LIN {X 0,Y 165.63,Z 443.538,A -85,B 0,C 180,E1 -26666.996,E2 -26666.996} C_VEL
LIN {X 0,Y 159.876,Z 456.557,A -85,B 0,C 180,E1 -26668.46,E2 -26668.46} C_VEL
LIN {X 0,Y 153.534,Z 468.796,A -85,B 0,C 180,E1 -26670.356,E2 -26670.356} C_VEL
LIN {X 0,Y 146.219,Z 480.711,A -85,B 0,C 180,E1 -26672.743,E2 -26672.743} C_VEL
LIN {X 0,Y 138.42,Z 491.702,A -85,B 0,C 180,E1 -26675.675,E2 -26675.675} C_VEL
LIN {X 0,Y 131.109,Z 500.936,A -85,B 0,C 180,E1 -26678.992,E2 -26678.992} C_VEL
LIN {X 0,Y 123.678,Z 509.508,A -85,B 0,C 180,E1 -26683.144,E2 -26683.144} C_VEL
LIN {X 0,Y 116.368,Z 517.34,A -85,B 0,C 180,E1 -26688.371,E2 -26688.371} C_VEL
LIN {X 0,Y 109.45,Z 524.137,A -85,B 0,C 180,E1 -26694.699,E2 -26694.699} C_VEL
LIN {X 0,Y 104.079,Z 529.404,A -85,B 0,C 180,E1 -26701.794,E2 -26701.794} C_VEL
LIN {X 0,Y 100.374,Z 533.276,A -85,B 0,C 180,E1 -26709.509,E2 -26709.509} C_VEL
LIN {X 0,Y 98.431,Z 535.839,A -85,B 0,C 180,E1 -26717.633,E2 -26717.633} C_VEL
LIN {X 0,Y 98.114,Z 537.142,A -85,B 0,C 180,E1 -26725.894,E2 -26725.894} C_VEL
LIN {X 0,Y 98.331,Z 537.315,A -85,B 0,C 180,E1 -26730.002,E2 -26730.002} C_VEL
LIN {X 0,Y 98.105,Z 537.113,A -85,B 0,C 180,E1 -26734.272,E2 -26734.272} C_VEL
LIN {X 0,Y 98.447,Z 535.805,A -85,B 0,C 180,E1 -26742.368,E2 -26742.368} C_VEL
LIN {X 0,Y 100.42,Z 533.218,A -85,B 0,C 180,E1 -26750.484,E2 -26750.484} C_VEL
LIN {X 0,Y 100.858,Z 532.685,A -85,B 0,C 180,E1 -26751.673,E2 -26751.673} C_VEL
LIN {X 0,Y 101.579,Z 531.255,A -85,B 0,C 180,E1 -26754.886,E2 -26754.886} C_VEL
LIN {X 0,Y 101.656,Z 528.502,A -85,B 0,C 180,E1 -26760.267,E2 -26760.267} C_VEL
LIN {X 0,Y 102.166,Z 525.971,A -85,B 0,C 180,E1 -26764.5,E2 -26764.5} C_VEL
LIN {X 0,Y 103.612,Z 523.788,A -85,B 0,C 180,E1 -26767.46,E2 -26767.46} C_VEL
LIN {X 0,Y 104.389,Z 523.002,A -85,B 0,C 180,E1 -26768.362,E2 -26768.362} C_VEL
LIN {X 0,Y 112.099,Z 515.87,A -85,B 0,C 180,E1 -26774.856,E2 -26774.856} C_VEL
LIN {X 0,Y 119.581,Z 508.219,A -85,B 0,C 180,E1 -26779.822,E2 -26779.822} C_VEL
LIN {X 0,Y 127.951,Z 498.926,A -85,B 0,C 180,E1 -26784.114,E2 -26784.114} C_VEL
LIN {X 0,Y 135.656,Z 489.398,A -85,B 0,C 180,E1 -26787.339,E2 -26787.339} C_VEL
LIN {X 0,Y 143.86,Z 477.978,A -85,B 0,C 180,E1 -26790.129,E2 -26790.129} C_VEL
LIN {X 0,Y 150.827,Z 466.569,A -85,B 0,C 180,E1 -26792.293,E2 -26792.293} C_VEL
LIN {X 0,Y 157.321,Z 454.193,A -85,B 0,C 180,E1 -26794.033,E2 -26794.033} C_VEL
LIN {X 0,Y 163.247,Z 440.627,A -85,B 0,C 180,E1 -26795.431,E2 -26795.431} C_VEL
LIN {X 0,Y 168.126,Z 426.606,A -85,B 0,C 180,E1 -26796.496,E2 -26796.496} C_VEL
LIN {X 0,Y 171.919,Z 412.179,A -85,B 0,C 180,E1 -26797.272,E2 -26797.272} C_VEL
LIN {X 0,Y 174.531,Z 397.305,A -85,B 0,C 180,E1 -26797.845,E2 -26797.845} C_VEL
LIN {X 0,Y 179.458,Z 349.439,A -85,B 0,C 180,E1 -26799.136,E2 -26799.136} C_VEL
LIN {X 0,Y 179.327,Z 348.411,A -85,B 0,C 180,E1 -26799.347,E2 -26799.347} C_VEL
LIN {X 0,Y 176.957,Z 341.677,A -85,B 0,C 180,E1 -26802.134,E2 -26802.134} C_VEL
LIN {X 0,Y 174.69,Z 335.913,A -85,B 0,C 180,E1 -26805.214,E2 -26805.214} C_VEL
LIN {X 0,Y 173.074,Z 332.046,A -85,B 0,C 180,E1 -26807.84,E2 -26807.84} C_VEL
LIN {X 0,Y 171.759,Z 329.073,A -85,B 0,C 180,E1 -26810.432,E2 -26810.432} C_VEL
LIN {X 0,Y 170.704,Z 326.371,A -85,B 0,C 180,E1 -26813.203,E2 -26813.203} C_VEL
LIN {X 0,Y 169.547,Z 323.722,A -85,B 0,C 180,E1 -26818.219,E2 -26818.219} C_VEL
LIN {X 0,Y 169.402,Z 323.159,A -85,B 0,C 180,E1 -26820,E2 -26820} C_VEL
LIN {X 0,Y 169.554,Z 323.797,A -85,B 0,C 180,E1 -26824.756,E2 -26824.756} C_VEL
LIN {X 0,Y 170.9,Z 326.862,A -85,B 0,C 180,E1 -26830.197,E2 -26830.197} C_VEL
LIN {X 0,Y 172.792,Z 331.172,A -85,B 0,C 180,E1 -26834.386,E2 -26834.386} C_VEL
LIN {X 0,Y 174.529,Z 335.32,A -85,B 0,C 180,E1 -26837.275,E2 -26837.275} C_VEL
LIN {X 0,Y 176.538,Z 340.227,A -85,B 0,C 180,E1 -26840.037,E2 -26840.037} C_VEL
LIN {X 0,Y 179.327,Z 347.998,A -85,B 0,C 180,E1 -26843.329,E2 -26843.329} C_VEL
LIN {X 0,Y 179.502,Z 348.597,A -85,B 0,C 180,E1 -26843.528,E2 -26843.528} C_VEL
LIN {X 0,Y 175.144,Z 392.557,A -85,B 0,C 180,E1 -26844.699,E2 -26844.699} C_VEL
LIN {X 0,Y 172.696,Z 407.451,A -85,B 0,C 180,E1 -26845.285,E2 -26845.285} C_VEL
LIN {X 0,Y 169.623,Z 420.1,A -85,B 0,C 180,E1 -26846.028,E2 -26846.028} C_VEL
LIN {X 0,Y 164.897,Z 434.553,A -85,B 0,C 180,E1 -26847.164,E2 -26847.164} C_VEL
LIN {X 0,Y 159.141,Z 448.284,A -85,B 0,C 180,E1 -26848.631,E2 -26848.631} C_VEL
LIN {X 0,Y 153.259,Z 459.955,A -85,B 0,C 180,E1 -26850.346,E2 -26850.346} C_VEL
LIN {X 0,Y 146.105,Z 471.975,A -85,B 0,C 180,E1 -26852.669,E2 -26852.669} C_VEL
LIN {X 0,Y 138.063,Z 483.246,A -85,B 0,C 180,E1 -26855.465,E2 -26855.465} C_VEL
LIN {X 0,Y 130.537,Z 492.568,A -85,B 0,C 180,E1 -26858.678,E2 -26858.678} C_VEL
LIN {X 0,Y 122.181,Z 501.604,A -85,B 0,C 180,E1 -26862.827,E2 -26862.827} C_VEL
LIN {X 0,Y 114.62,Z 508.971,A -85,B 0,C 180,E1 -26867.586,E2 -26867.586} C_VEL
LIN {X 0,Y 108.945,Z 514.139,A -85,B 0,C 180,E1 -26872.204,E2 -26872.204} C_VEL
LIN {X 0,Y 102.132,Z 519.688,A -85,B 0,C 180,E1 -26878.928,E2 -26878.928} C_VEL
LIN {X 0,Y 98.187,Z 522.898,A -85,B 0,C 180,E1 -26884.565,E2 -26884.565} C_VEL
LIN {X 0,Y 94.287,Z 525.978,A -85,B 0,C 180,E1 -26892.652,E2 -26892.652} C_VEL
LIN {X 0,Y 92.052,Z 527.802,A -85,B 0,C 180,E1 -26901.215,E2 -26901.215} C_VEL
LIN {X 0,Y 91.365,Z 528.414,A -85,B 0,C 180,E1 -26909.998,E2 -26909.998} C_VEL
LIN {X 0,Y 92.006,Z 527.836,A -85,B 0,C 180,E1 -26918.786,E2 -26918.786} C_VEL
LIN {X 0,Y 94.227,Z 526.051,A -85,B 0,C 180,E1 -26927.356,E2 -26927.356} C_VEL
LIN {X 0,Y 98.143,Z 523.004,A -85,B 0,C 180,E1 -26935.444,E2 -26935.444} C_VEL
LIN {X 0,Y 103.601,Z 518.617,A -85,B 0,C 180,E1 -26942.865,E2 -26942.865} C_VEL
LIN {X 0,Y 110.742,Z 512.748,A -85,B 0,C 180,E1 -26949.39,E2 -26949.39} C_VEL
LIN {X 0,Y 117.572,Z 506.34,A -85,B 0,C 180,E1 -26954.495,E2 -26954.495} C_VEL
LIN {X 0,Y 125.598,Z 498.252,A -85,B 0,C 180,E1 -26959.059,E2 -26959.059} C_VEL
LIN {X 0,Y 134.204,Z 488.494,A -85,B 0,C 180,E1 -26962.995,E2 -26962.995} C_VEL
LIN {X 0,Y 141.959,Z 478.341,A -85,B 0,C 180,E1 -26966.019,E2 -26966.019} C_VEL
LIN {X 0,Y 149.557,Z 466.932,A -85,B 0,C 180,E1 -26968.501,E2 -26968.501} C_VEL
LIN {X 0,Y 156.253,Z 454.749,A -85,B 0,C 180,E1 -26970.625,E2 -26970.625} C_VEL
LIN {X 0,Y 161.922,Z 442.664,A -85,B 0,C 180,E1 -26972.168,E2 -26972.168} C_VEL
LIN {X 0,Y 166.986,Z 429.457,A -85,B 0,C 180,E1 -26973.423,E2 -26973.423} C_VEL
LIN {X 0,Y 171.178,Z 415.274,A -85,B 0,C 180,E1 -26974.414,E2 -26974.414} C_VEL
LIN {X 0,Y 174.201,Z 400.761,A -85,B 0,C 180,E1 -26975.152,E2 -26975.152} C_VEL
LIN {X 0,Y 176.229,Z 385.179,A -85,B 0,C 180,E1 -26975.622,E2 -26975.622} C_VEL
LIN {X 0,Y 179.732,Z 348.839,A -85,B 0,C 180,E1 -26976.589,E2 -26976.589} C_VEL
LIN {X 0,Y 177.194,Z 341.617,A -85,B 0,C 180,E1 -26979.561,E2 -26979.561} C_VEL
LIN {X 0,Y 175.174,Z 336.455,A -85,B 0,C 180,E1 -26982.287,E2 -26982.287} C_VEL
LIN {X 0,Y 173.214,Z 331.803,A -85,B 0,C 180,E1 -26985.46,E2 -26985.46} C_VEL
LIN {X 0,Y 172.172,Z 329.574,A -85,B 0,C 180,E1 -26987.488,E2 -26987.488} C_VEL
LIN {X 0,Y 170.897,Z 326.546,A -85,B 0,C 180,E1 -26990.773,E2 -26990.773} C_VEL
LIN {X 0,Y 169.875,Z 324.156,A -85,B 0,C 180,E1 -26995.253,E2 -26995.253} C_VEL
LIN {X 0,Y 169.668,Z 323.599,A -85,B 0,C 180,E1 -26997.626,E2 -26997.626} C_VEL
LIN {X 0,Y 169.698,Z 323.594,A -85,B 0,C 180,E1 -27000.296,E2 -27000.296} C_VEL
LIN {X 0,Y 170.29,Z 325.277,A -85,B 0,C 180,E1 -27004.438,E2 -27004.438} C_VEL
LIN {X 0,Y 171.166,Z 327.18,A -85,B 0,C 180,E1 -27007.372,E2 -27007.372} C_VEL
LIN {X 0,Y 172.943,Z 331.435,A -85,B 0,C 180,E1 -27011.426,E2 -27011.426} C_VEL
LIN {X 0,Y 174.487,Z 335.046,A -85,B 0,C 180,E1 -27014.059,E2 -27014.059} C_VEL
LIN {X 0,Y 176.715,Z 340.576,A -85,B 0,C 180,E1 -27017.205,E2 -27017.205} C_VEL
LIN {X 0,Y 179.259,Z 347.708,A -85,B 0,C 180,E1 -27020.287,E2 -27020.287} C_VEL
LIN {X 0,Y 179.732,Z 349.271,A -85,B 0,C 180,E1 -27020.831,E2 -27020.831} C_VEL
LIN {X 0,Y 174.564,Z 399.199,A -85,B 0,C 180,E1 -27022.187,E2 -27022.187} C_VEL
LIN {X 0,Y 171.726,Z 414.147,A -85,B 0,C 180,E1 -27022.768,E2 -27022.768} C_VEL
LIN {X 0,Y 167.744,Z 428.611,A -85,B 0,C 180,E1 -27023.584,E2 -27023.584} C_VEL
LIN {X 0,Y 162.524,Z 443.079,A -85,B 0,C 180,E1 -27024.76,E2 -27024.76} C_VEL
LIN {X 0,Y 156.61,Z 456.14,A -85,B 0,C 180,E1 -27026.17,E2 -27026.17} C_VEL
LIN {X 0,Y 150.038,Z 468.405,A -85,B 0,C 180,E1 -27027.993,E2 -27027.993} C_VEL
LIN {X 0,Y 142.493,Z 480.341,A -85,B 0,C 180,E1 -27030.333,E2 -27030.333} C_VEL
LIN {X 0,Y 134.362,Z 491.343,A -85,B 0,C 180,E1 -27033.189,E2 -27033.189} C_VEL
LIN {X 0,Y 126.712,Z 500.585,A -85,B 0,C 180,E1 -27036.467,E2 -27036.467} C_VEL
LIN {X 0,Y 118.259,Z 509.78,A -85,B 0,C 180,E1 -27040.975,E2 -27040.975} C_VEL
LIN {X 0,Y 111.092,Z 516.998,A -85,B 0,C 180,E1 -27045.904,E2 -27045.904} C_VEL
LIN {X 0,Y 103.658,Z 523.798,A -85,B 0,C 180,E1 -27052.398,E2 -27052.398} C_VEL
LIN {X 0,Y 97.793,Z 529.066,A -85,B 0,C 180,E1 -27059.8,E2 -27059.8} C_VEL
LIN {X 0,Y 93.682,Z 532.94,A -85,B 0,C 180,E1 -27067.972,E2 -27067.972} C_VEL
LIN {X 0,Y 91.456,Z 535.504,A -85,B 0,C 180,E1 -27076.673,E2 -27076.673} C_VEL
LIN {X 0,Y 91.004,Z 536.808,A -85,B 0,C 180,E1 -27085.573,E2 -27085.573} C_VEL
LIN {X 0,Y 91.223,Z 536.982,A -85,B 0,C 180,E1 -27090.002,E2 -27090.002} C_VEL
LIN {X 0,Y 91.006,Z 536.799,A -85,B 0,C 180,E1 -27094.431,E2 -27094.431} C_VEL
LIN {X 0,Y 91.471,Z 535.469,A -85,B 0,C 180,E1 -27103.328,E2 -27103.328} C_VEL
LIN {X 0,Y 93.942,Z 532.637,A -85,B 0,C 180,E1 -27112.6,E2 -27112.6} C_VEL
LIN {X 0,Y 98.235,Z 528.616,A -85,B 0,C 180,E1 -27120.852,E2 -27120.852} C_VEL
LIN {X 0,Y 104.389,Z 523.002,A -85,B 0,C 180,E1 -27128.362,E2 -27128.362} C_VEL
LIN {X 0,Y 106.483,Z 520.606,A -85,B 0,C 180,E1 -27131.065,E2 -27131.065} C_VEL
LIN {X 0,Y 108.822,Z 516.381,A -85,B 0,C 180,E1 -27135.684,E2 -27135.684} C_VEL
LIN {X 0,Y 111.632,Z 511.724,A -85,B 0,C 180,E1 -27140.005,E2 -27140.005} C_VEL
LIN {X 0,Y 114.344,Z 508.588,A -85,B 0,C 180,E1 -27142.15,E2 -27142.15} C_VEL
LIN {X 0,Y 122.587,Z 500.012,A -85,B 0,C 180,E1 -27146.233,E2 -27146.233} C_VEL
LIN {X 0,Y 130.553,Z 490.711,A -85,B 0,C 180,E1 -27149.466,E2 -27149.466} C_VEL
LIN {X 0,Y 139.016,Z 479.648,A -85,B 0,C 180,E1 -27152.217,E2 -27152.217} C_VEL
LIN {X 0,Y 146.943,Z 467.351,A -85,B 0,C 180,E1 -27154.558,E2 -27154.558} C_VEL
LIN {X 0,Y 153.578,Z 455.24,A -85,B 0,C 180,E1 -27156.24,E2 -27156.24} C_VEL
LIN {X 0,Y 159.655,Z 442.016,A -85,B 0,C 180,E1 -27157.581,E2 -27157.581} C_VEL
LIN {X 0,Y 164.638,Z 428.465,A -85,B 0,C 180,E1 -27158.611,E2 -27158.611} C_VEL
LIN {X 0,Y 168.878,Z 413.351,A -85,B 0,C 180,E1 -27159.419,E2 -27159.419} C_VEL
LIN {X 0,Y 171.751,Z 397.879,A -85,B 0,C 180,E1 -27160.002,E2 -27160.002} C_VEL
LIN {X 0,Y 176.586,Z 352.392,A -85,B 0,C 180,E1 -27161.19,E2 -27161.19} C_VEL
LIN {X 0,Y 174.45,Z 345.846,A -85,B 0,C 180,E1 -27164.071,E2 -27164.071} C_VEL
LIN {X 0,Y 172.065,Z 339.511,A -85,B 0,C 180,E1 -27167.917,E2 -27167.917} C_VEL
LIN {X 0,Y 170.658,Z 336.056,A -85,B 0,C 180,E1 -27170.818,E2 -27170.818} C_VEL
LIN {X 0,Y 169.526,Z 333.041,A -85,B 0,C 180,E1 -27174.051,E2 -27174.051} C_VEL
LIN {X 0,Y 168.609,Z 330.633,A -85,B 0,C 180,E1 -27178.806,E2 -27178.806} C_VEL
LIN {X 0,Y 168.533,Z 330.233,A -85,B 0,C 180,E1 -27180,E2 -27180} C_VEL
LIN {X 0,Y 168.624,Z 330.752,A -85,B 0,C 180,E1 -27184.283,E2 -27184.283} C_VEL
LIN {X 0,Y 169.777,Z 333.605,A -85,B 0,C 180,E1 -27189.531,E2 -27189.531} C_VEL
LIN {X 0,Y 171.5,Z 337.856,A -85,B 0,C 180,E1 -27193.705,E2 -27193.705} C_VEL
LIN {X 0,Y 173.35,Z 342.671,A -85,B 0,C 180,E1 -27196.989,E2 -27196.989} C_VEL
LIN {X 0,Y 175.206,Z 347.777,A -85,B 0,C 180,E1 -27199.681,E2 -27199.681} C_VEL
LIN {X 0,Y 176.615,Z 352.119,A -85,B 0,C 180,E1 -27201.51,E2 -27201.51} C_VEL
LIN {X 0,Y 171.973,Z 396.261,A -85,B 0,C 180,E1 -27202.65,E2 -27202.65} C_VEL
LIN {X 0,Y 169.092,Z 411.279,A -85,B 0,C 180,E1 -27203.27,E2 -27203.27} C_VEL
LIN {X 0,Y 165.171,Z 425.566,A -85,B 0,C 180,E1 -27204.194,E2 -27204.194} C_VEL
LIN {X 0,Y 160.331,Z 438.781,A -85,B 0,C 180,E1 -27205.299,E2 -27205.299} C_VEL
LIN {X 0,Y 154.397,Z 451.68,A -85,B 0,C 180,E1 -27206.707,E2 -27206.707} C_VEL
LIN {X 0,Y 147.791,Z 463.904,A -85,B 0,C 180,E1 -27208.646,E2 -27208.646} C_VEL
LIN {X 0,Y 141.006,Z 474.391,A -85,B 0,C 180,E1 -27210.708,E2 -27210.708} C_VEL
LIN {X 0,Y 132.761,Z 485.257,A -85,B 0,C 180,E1 -27213.512,E2 -27213.512} C_VEL
LIN {X 0,Y 124.974,Z 494.32,A -85,B 0,C 180,E1 -27216.739,E2 -27216.739} C_VEL
LIN {X 0,Y 116.278,Z 503.071,A -85,B 0,C 180,E1 -27220.929,E2 -27220.929} C_VEL
LIN {X 0,Y 109.458,Z 509.315,A -85,B 0,C 180,E1 -27225.066,E2 -27225.066} C_VEL
LIN {X 0,Y 103.435,Z 514.475,A -85,B 0,C 180,E1 -27229.797,E2 -27229.797} C_VEL
LIN {X 0,Y 96.114,Z 520.023,A -85,B 0,C 180,E1 -27236.741,E2 -27236.741} C_VEL
LIN {X 0,Y 91.807,Z 523.233,A -85,B 0,C 180,E1 -27242.656,E2 -27242.656} C_VEL
LIN {X 0,Y 87.54,Z 526.311,A -85,B 0,C 180,E1 -27251.267,E2 -27251.267} C_VEL
LIN {X 0,Y 85.068,Z 528.134,A -85,B 0,C 180,E1 -27260.488,E2 -27260.488} C_VEL
LIN {X 0,Y 84.3,Z 528.746,A -85,B 0,C 180,E1 -27269.998,E2 -27269.998} C_VEL
LIN {X 0,Y 84.994,Z 528.168,A -85,B 0,C 180,E1 -27279.517,E2 -27279.517} C_VEL
LIN {X 0,Y 87.49,Z 526.383,A -85,B 0,C 180,E1 -27288.741,E2 -27288.741} C_VEL
LIN {X 0,Y 91.766,Z 523.338,A -85,B 0,C 180,E1 -27297.354,E2 -27297.354} C_VEL
LIN {X 0,Y 97.719,Z 518.949,A -85,B 0,C 180,E1 -27305.123,E2 -27305.123} C_VEL
LIN {X 0,Y 105.331,Z 513.084,A -85,B 0,C 180,E1 -27311.851,E2 -27311.851} C_VEL
LIN {X 0,Y 112.614,Z 506.677,A -85,B 0,C 180,E1 -27317.029,E2 -27317.029} C_VEL
LIN {X 0,Y 119.808,Z 499.813,A -85,B 0,C 180,E1 -27321.007,E2 -27321.007} C_VEL
LIN {X 0,Y 127.457,Z 491.798,A -85,B 0,C 180,E1 -27324.418,E2 -27324.418} C_VEL
LIN {X 0,Y 135.392,Z 482.257,A -85,B 0,C 180,E1 -27327.51,E2 -27327.51} C_VEL
LIN {X 0,Y 143.696,Z 470.728,A -85,B 0,C 180,E1 -27330.239,E2 -27330.239} C_VEL
LIN {X 0,Y 149.988,Z 460.498,A -85,B 0,C 180,E1 -27332.108,E2 -27332.108} C_VEL
LIN {X 0,Y 156.542,Z 447.881,A -85,B 0,C 180,E1 -27333.88,E2 -27333.88} C_VEL
LIN {X 0,Y 161.735,Z 435.963,A -85,B 0,C 180,E1 -27335.103,E2 -27335.103} C_VEL
LIN {X 0,Y 166.192,Z 423.162,A -85,B 0,C 180,E1 -27336.129,E2 -27336.129} C_VEL
LIN {X 0,Y 169.968,Z 408.622,A -85,B 0,C 180,E1 -27336.989,E2 -27336.989} C_VEL
LIN {X 0,Y 172.529,Z 394.256,A -85,B 0,C 180,E1 -27337.533,E2 -27337.533} C_VEL
LIN {X 0,Y 176.858,Z 352.376,A -85,B 0,C 180,E1 -27338.606,E2 -27338.606} C_VEL
LIN {X 0,Y 174.75,Z 345.892,A -85,B 0,C 180,E1 -27341.448,E2 -27341.448} C_VEL
LIN {X 0,Y 172.472,Z 339.853,A -85,B 0,C 180,E1 -27345.094,E2 -27345.094} C_VEL
LIN {X 0,Y 171.056,Z 336.449,A -85,B 0,C 180,E1 -27347.95,E2 -27347.95} C_VEL
LIN {X 0,Y 169.834,Z 333.379,A -85,B 0,C 180,E1 -27351.346,E2 -27351.346} C_VEL
LIN {X 0,Y 168.939,Z 331.064,A -85,B 0,C 180,E1 -27355.825,E2 -27355.825} C_VEL
LIN {X 0,Y 168.799,Z 330.627,A -85,B 0,C 180,E1 -27357.734,E2 -27357.734} C_VEL
LIN {X 0,Y 168.845,Z 330.755,A -85,B 0,C 180,E1 -27360.596,E2 -27360.596} C_VEL
LIN {X 0,Y 169.404,Z 332.428,A -85,B 0,C 180,E1 -27364.461,E2 -27364.461} C_VEL
LIN {X 0,Y 170.113,Z 334.141,A -85,B 0,C 180,E1 -27366.97,E2 -27366.97} C_VEL
LIN {X 0,Y 171.58,Z 337.97,A -85,B 0,C 180,E1 -27370.62,E2 -27370.62} C_VEL
LIN {X 0,Y 173.094,Z 341.842,A -85,B 0,C 180,E1 -27373.426,E2 -27373.426} C_VEL
LIN {X 0,Y 174.997,Z 346.976,A -85,B 0,C 180,E1 -27376.327,E2 -27376.327} C_VEL
LIN {X 0,Y 176.805,Z 352.535,A -85,B 0,C 180,E1 -27378.75,E2 -27378.75} C_VEL
LIN {X 0,Y 171.814,Z 399.481,A -85,B 0,C 180,E1 -27380.032,E2 -27380.032} C_VEL
LIN {X 0,Y 168.901,Z 414.27,A -85,B 0,C 180,E1 -27380.577,E2 -27380.577} C_VEL
LIN {X 0,Y 164.64,Z 429.218,A -85,B 0,C 180,E1 -27381.396,E2 -27381.396} C_VEL
LIN {X 0,Y 159.681,Z 442.622,A -85,B 0,C 180,E1 -27382.446,E2 -27382.446} C_VEL
LIN {X 0,Y 153.605,Z 455.724,A -85,B 0,C 180,E1 -27383.788,E2 -27383.788} C_VEL
LIN {X 0,Y 146.861,Z 467.937,A -85,B 0,C 180,E1 -27385.511,E2 -27385.511} C_VEL
LIN {X 0,Y 139.023,Z 479.97,A -85,B 0,C 180,E1 -27387.792,E2 -27387.792} C_VEL
LIN {X 0,Y 130.578,Z 490.985,A -85,B 0,C 180,E1 -27390.557,E2 -27390.557} C_VEL
LIN {X 0,Y 122.594,Z 500.236,A -85,B 0,C 180,E1 -27393.776,E2 -27393.776} C_VEL
LIN {X 0,Y 114.196,Z 508.969,A -85,B 0,C 180,E1 -27397.982,E2 -27397.982} C_VEL
LIN {X 0,Y 106.046,Z 516.658,A -85,B 0,C 180,E1 -27403.2,E2 -27403.2} C_VEL
LIN {X 0,Y 98.064,Z 523.459,A -85,B 0,C 180,E1 -27409.837,E2 -27409.837} C_VEL
LIN {X 0,Y 91.665,Z 528.729,A -85,B 0,C 180,E1 -27417.544,E2 -27417.544} C_VEL
LIN {X 0,Y 87.075,Z 532.603,A -85,B 0,C 180,E1 -27426.201,E2 -27426.201} C_VEL
LIN {X 0,Y 84.485,Z 535.168,A -85,B 0,C 180,E1 -27435.551,E2 -27435.551} C_VEL
LIN {X 0,Y 83.899,Z 536.473,A -85,B 0,C 180,E1 -27445.197,E2 -27445.197} C_VEL
LIN {X 0,Y 84.133,Z 536.649,A -85,B 0,C 180,E1 -27450.002,E2 -27450.002} C_VEL
LIN {X 0,Y 83.9,Z 536.464,A -85,B 0,C 180,E1 -27454.807,E2 -27454.807} C_VEL
LIN {X 0,Y 84.501,Z 535.132,A -85,B 0,C 180,E1 -27464.45,E2 -27464.45} C_VEL
LIN {X 0,Y 87.109,Z 532.543,A -85,B 0,C 180,E1 -27473.793,E2 -27473.793} C_VEL
LIN {X 0,Y 91.722,Z 528.594,A -85,B 0,C 180,E1 -27482.559,E2 -27482.559} C_VEL
LIN {X 0,Y 98.26,Z 523.174,A -85,B 0,C 180,E1 -27490.364,E2 -27490.364} C_VEL
LIN {X 0,Y 106.041,Z 516.504,A -85,B 0,C 180,E1 -27496.807,E2 -27496.807} C_VEL
LIN {X 0,Y 114.344,Z 508.588,A -85,B 0,C 180,E1 -27502.15,E2 -27502.15} C_VEL
LIN {X 0,Y 117.141,Z 505.31,A -85,B 0,C 180,E1 -27504.162,E2 -27504.162} C_VEL
LIN {X 0,Y 120.678,Z 499.746,A -85,B 0,C 180,E1 -27507.746,E2 -27507.746} C_VEL
LIN {X 0,Y 124.469,Z 493.764,A -85,B 0,C 180,E1 -27510.974,E2 -27510.974} C_VEL
LIN {X 0,Y 127.526,Z 489.803,A -85,B 0,C 180,E1 -27512.4,E2 -27512.4} C_VEL
LIN {X 0,Y 136.568,Z 478.275,A -85,B 0,C 180,E1 -27515.096,E2 -27515.096} C_VEL
LIN {X 0,Y 144.752,Z 465.749,A -85,B 0,C 180,E1 -27517.293,E2 -27517.293} C_VEL
LIN {X 0,Y 151.616,Z 453.301,A -85,B 0,C 180,E1 -27518.888,E2 -27518.888} C_VEL
LIN {X 0,Y 157.856,Z 439.627,A -85,B 0,C 180,E1 -27520.139,E2 -27520.139} C_VEL
LIN {X 0,Y 162.577,Z 426.731,A -85,B 0,C 180,E1 -27521.02,E2 -27521.02} C_VEL
LIN {X 0,Y 166.588,Z 412.267,A -85,B 0,C 180,E1 -27521.728,E2 -27521.728} C_VEL
LIN {X 0,Y 169.431,Z 396.965,A -85,B 0,C 180,E1 -27522.25,E2 -27522.25} C_VEL
LIN {X 0,Y 173.884,Z 355.821,A -85,B 0,C 180,E1 -27523.313,E2 -27523.313} C_VEL
LIN {X 0,Y 172.125,Z 350.295,A -85,B 0,C 180,E1 -27526.046,E2 -27526.046} C_VEL
LIN {X 0,Y 170.39,Z 345.291,A -85,B 0,C 180,E1 -27529.304,E2 -27529.304} C_VEL
LIN {X 0,Y 169.28,Z 342.309,A -85,B 0,C 180,E1 -27531.946,E2 -27531.946} C_VEL
LIN {X 0,Y 168.467,Z 339.868,A -85,B 0,C 180,E1 -27534.614,E2 -27534.614} C_VEL
LIN {X 0,Y 167.733,Z 337.709,A -85,B 0,C 180,E1 -27538.8,E2 -27538.8} C_VEL
LIN {X 0,Y 167.663,Z 337.292,A -85,B 0,C 180,E1 -27540,E2 -27540} C_VEL
LIN {X 0,Y 167.755,Z 337.788,A -85,B 0,C 180,E1 -27544.194,E2 -27544.194} C_VEL
LIN {X 0,Y 168.713,Z 340.446,A -85,B 0,C 180,E1 -27548.988,E2 -27548.988} C_VEL
LIN {X 0,Y 170.202,Z 344.537,A -85,B 0,C 180,E1 -27552.977,E2 -27552.977} C_VEL
LIN {X 0,Y 172.076,Z 349.751,A -85,B 0,C 180,E1 -27556.537,E2 -27556.537} C_VEL
LIN {X 0,Y 173.931,Z 355.662,A -85,B 0,C 180,E1 -27559.414,E2 -27559.414} C_VEL
LIN {X 0,Y 169.481,Z 396.544,A -85,B 0,C 180,E1 -27560.423,E2 -27560.423} C_VEL
LIN {X 0,Y 166.581,Z 411.332,A -85,B 0,C 180,E1 -27561.006,E2 -27561.006} C_VEL
LIN {X 0,Y 162.78,Z 424.977,A -85,B 0,C 180,E1 -27561.835,E2 -27561.835} C_VEL
LIN {X 0,Y 158.185,Z 437.489,A -85,B 0,C 180,E1 -27562.794,E2 -27562.794} C_VEL
LIN {X 0,Y 152.11,Z 450.684,A -85,B 0,C 180,E1 -27564.144,E2 -27564.144} C_VEL
LIN {X 0,Y 145.867,Z 462.102,A -85,B 0,C 180,E1 -27565.784,E2 -27565.784} C_VEL
LIN {X 0,Y 138.258,Z 473.788,A -85,B 0,C 180,E1 -27567.967,E2 -27567.967} C_VEL
LIN {X 0,Y 130.344,Z 483.981,A -85,B 0,C 180,E1 -27570.378,E2 -27570.378} C_VEL
LIN {X 0,Y 122.165,Z 493.28,A -85,B 0,C 180,E1 -27573.47,E2 -27573.47} C_VEL
LIN {X 0,Y 112.996,Z 502.299,A -85,B 0,C 180,E1 -27577.531,E2 -27577.531} C_VEL
LIN {X 0,Y 104.54,Z 509.658,A -85,B 0,C 180,E1 -27582.31,E2 -27582.31} C_VEL
LIN {X 0,Y 98.128,Z 514.813,A -85,B 0,C 180,E1 -27587.124,E2 -27587.124} C_VEL
LIN {X 0,Y 90.261,Z 520.359,A -85,B 0,C 180,E1 -27594.268,E2 -27594.268} C_VEL
LIN {X 0,Y 85.553,Z 523.567,A -85,B 0,C 180,E1 -27600.468,E2 -27600.468} C_VEL
LIN {X 0,Y 80.862,Z 526.644,A -85,B 0,C 180,E1 -27609.654,E2 -27609.654} C_VEL
LIN {X 0,Y 78.072,Z 528.467,A -85,B 0,C 180,E1 -27619.626,E2 -27619.626} C_VEL
LIN {X 0,Y 77.225,Z 529.078,A -85,B 0,C 180,E1 -27629.998,E2 -27629.998} C_VEL
LIN {X 0,Y 78.014,Z 528.5,A -85,B 0,C 180,E1 -27640.378,E2 -27640.378} C_VEL
LIN {X 0,Y 80.793,Z 526.716,A -85,B 0,C 180,E1 -27650.36,E2 -27650.36} C_VEL
LIN {X 0,Y 85.515,Z 523.67,A -85,B 0,C 180,E1 -27659.543,E2 -27659.543} C_VEL
LIN {X 0,Y 92.011,Z 519.282,A -85,B 0,C 180,E1 -27667.663,E2 -27667.663} C_VEL
LIN {X 0,Y 100.136,Z 513.42,A -85,B 0,C 180,E1 -27674.572,E2 -27674.572} C_VEL
LIN {X 0,Y 108.02,Z 506.916,A -85,B 0,C 180,E1 -27679.857,E2 -27679.857} C_VEL
LIN {X 0,Y 116.797,Z 498.936,A -85,B 0,C 180,E1 -27684.321,E2 -27684.321} C_VEL
LIN {X 0,Y 126.185,Z 489.2,A -85,B 0,C 180,E1 -27688.139,E2 -27688.139} C_VEL
LIN {X 0,Y 134.554,Z 479.072,A -85,B 0,C 180,E1 -27691.027,E2 -27691.027} C_VEL
LIN {X 0,Y 142.496,Z 467.975,A -85,B 0,C 180,E1 -27693.31,E2 -27693.31} C_VEL
LIN {X 0,Y 149.814,Z 455.577,A -85,B 0,C 180,E1 -27695.351,E2 -27695.351} C_VEL
LIN {X 0,Y 155.822,Z 443.569,A -85,B 0,C 180,E1 -27696.772,E2 -27696.772} C_VEL
LIN {X 0,Y 161.543,Z 429.372,A -85,B 0,C 180,E1 -27697.999,E2 -27697.999} C_VEL
LIN {X 0,Y 165.974,Z 414.934,A -85,B 0,C 180,E1 -27698.909,E2 -27698.909} C_VEL
LIN {X 0,Y 169.028,Z 400.886,A -85,B 0,C 180,E1 -27699.558,E2 -27699.558} C_VEL
LIN {X 0,Y 171.273,Z 384.215,A -85,B 0,C 180,E1 -27700.006,E2 -27700.006} C_VEL
LIN {X 0,Y 174.184,Z 355.781,A -85,B 0,C 180,E1 -27700.729,E2 -27700.729} C_VEL
LIN {X 0,Y 172.281,Z 349.813,A -85,B 0,C 180,E1 -27703.712,E2 -27703.712} C_VEL
LIN {X 0,Y 170.483,Z 344.736,A -85,B 0,C 180,E1 -27707.176,E2 -27707.176} C_VEL
LIN {X 0,Y 168.886,Z 340.389,A -85,B 0,C 180,E1 -27711.59,E2 -27711.59} C_VEL
LIN {X 0,Y 168.071,Z 338.153,A -85,B 0,C 180,E1 -27715.803,E2 -27715.803} C_VEL
LIN {X 0,Y 167.935,Z 337.725,A -85,B 0,C 180,E1 -27717.601,E2 -27717.601} C_VEL
LIN {X 0,Y 167.976,Z 337.835,A -85,B 0,C 180,E1 -27720.599,E2 -27720.599} C_VEL
LIN {X 0,Y 168.587,Z 339.766,A -85,B 0,C 180,E1 -27724.782,E2 -27724.782} C_VEL
LIN {X 0,Y 169.101,Z 341.329,A -85,B 0,C 180,E1 -27726.712,E2 -27726.712} C_VEL
LIN {X 0,Y 170.252,Z 344.508,A -85,B 0,C 180,E1 -27729.804,E2 -27729.804} C_VEL
LIN {X 0,Y 171.566,Z 348.184,A -85,B 0,C 180,E1 -27732.494,E2 -27732.494} C_VEL
LIN {X 0,Y 173.345,Z 353.543,A -85,B 0,C 180,E1 -27735.482,E2 -27735.482} C_VEL
LIN {X 0,Y 174.133,Z 356.068,A -85,B 0,C 180,E1 -27736.655,E2 -27736.655} C_VEL
LIN {X 0,Y 169.349,Z 399.51,A -85,B 0,C 180,E1 -27737.795,E2 -27737.795} C_VEL
LIN {X 0,Y 166.34,Z 414.353,A -85,B 0,C 180,E1 -27738.312,E2 -27738.312} C_VEL
LIN {X 0,Y 162.182,Z 428.694,A -85,B 0,C 180,E1 -27739.057,E2 -27739.057} C_VEL
LIN {X 0,Y 157.105,Z 442.164,A -85,B 0,C 180,E1 -27740.05,E2 -27740.05} C_VEL
LIN {X 0,Y 150.863,Z 455.306,A -85,B 0,C 180,E1 -27741.302,E2 -27741.302} C_VEL
LIN {X 0,Y 144.057,Z 467.329,A -85,B 0,C 180,E1 -27742.9,E2 -27742.9} C_VEL
LIN {X 0,Y 135.836,Z 479.599,A -85,B 0,C 180,E1 -27745.123,E2 -27745.123} C_VEL
LIN {X 0,Y 127.087,Z 490.627,A -85,B 0,C 180,E1 -27747.776,E2 -27747.776} C_VEL
LIN {X 0,Y 118.755,Z 499.887,A -85,B 0,C 180,E1 -27750.898,E2 -27750.898} C_VEL
LIN {X 0,Y 110.875,Z 507.726,A -85,B 0,C 180,E1 -27754.514,E2 -27754.514} C_VEL
LIN {X 0,Y 103.539,Z 514.322,A -85,B 0,C 180,E1 -27758.688,E2 -27758.688} C_VEL
LIN {X 0,Y 94.695,Z 521.569,A -85,B 0,C 180,E1 -27765.168,E2 -27765.168} C_VEL
LIN {X 0,Y 87.282,Z 527.215,A -85,B 0,C 180,E1 -27772.853,E2 -27772.853} C_VEL
LIN {X 0,Y 82.898,Z 530.499,A -85,B 0,C 180,E1 -27779.427,E2 -27779.427} C_VEL
LIN {X 0,Y 78.742,Z 533.707,A -85,B 0,C 180,E1 -27789.085,E2 -27789.085} C_VEL
LIN {X 0,Y 76.928,Z 535.642,A -85,B 0,C 180,E1 -27799.474,E2 -27799.474} C_VEL
LIN {X 0,Y 76.79,Z 536.139,A -85,B 0,C 180,E1 -27804.751,E2 -27804.751} C_VEL
LIN {X 0,Y 77.047,Z 536.316,A -85,B 0,C 180,E1 -27810.002,E2 -27810.002} C_VEL
LIN {X 0,Y 76.793,Z 536.13,A -85,B 0,C 180,E1 -27815.253,E2 -27815.253} C_VEL
LIN {X 0,Y 77.573,Z 534.795,A -85,B 0,C 180,E1 -27825.773,E2 -27825.773} C_VEL
LIN {X 0,Y 80.599,Z 532.206,A -85,B 0,C 180,E1 -27835.85,E2 -27835.85} C_VEL
LIN {X 0,Y 85.67,Z 528.305,A -85,B 0,C 180,E1 -27845.049,E2 -27845.049} C_VEL
LIN {X 0,Y 92.675,Z 523.003,A -85,B 0,C 180,E1 -27853.042,E2 -27853.042} C_VEL
LIN {X 0,Y 101.264,Z 516.161,A -85,B 0,C 180,E1 -27859.769,E2 -27859.769} C_VEL
LIN {X 0,Y 109.317,Z 508.933,A -85,B 0,C 180,E1 -27864.706,E2 -27864.706} C_VEL
LIN {X 0,Y 117.395,Z 501.029,A -85,B 0,C 180,E1 -27868.551,E2 -27868.551} C_VEL
LIN {X 0,Y 125.662,Z 491.994,A -85,B 0,C 180,E1 -27871.748,E2 -27871.748} C_VEL
LIN {X 0,Y 127.526,Z 489.803,A -85,B 0,C 180,E1 -27872.4,E2 -27872.4} C_VEL
LIN {X 0,Y 130.56,Z 485.712,A -85,B 0,C 180,E1 -27873.738,E2 -27873.738} C_VEL
LIN {X 0,Y 134.41,Z 478.89,A -85,B 0,C 180,E1 -27876.383,E2 -27876.383} C_VEL
LIN {X 0,Y 138.22,Z 471.768,A -85,B 0,C 180,E1 -27878.777,E2 -27878.777} C_VEL
LIN {X 0,Y 141.066,Z 467.061,A -85,B 0,C 180,E1 -27879.715,E2 -27879.715} C_VEL
LIN {X 0,Y 148.409,Z 454.388,A -85,B 0,C 180,E1 -27881.283,E2 -27881.283} C_VEL
LIN {X 0,Y 154.783,Z 441.075,A -85,B 0,C 180,E1 -27882.462,E2 -27882.462} C_VEL
LIN {X 0,Y 159.998,Z 427.387,A -85,B 0,C 180,E1 -27883.361,E2 -27883.361} C_VEL
LIN {X 0,Y 164.173,Z 412.97,A -85,B 0,C 180,E1 -27884.022,E2 -27884.022} C_VEL
LIN {X 0,Y 166.985,Z 398.735,A -85,B 0,C 180,E1 -27884.516,E2 -27884.516} C_VEL
LIN {X 0,Y 171.416,Z 359.622,A -85,B 0,C 180,E1 -27885.457,E2 -27885.457} C_VEL
LIN {X 0,Y 169.854,Z 354.388,A -85,B 0,C 180,E1 -27888.363,E2 -27888.363} C_VEL
LIN {X 0,Y 168.539,Z 350.141,A -85,B 0,C 180,E1 -27891.457,E2 -27891.457} C_VEL
LIN {X 0,Y 167.421,Z 346.721,A -85,B 0,C 180,E1 -27895.184,E2 -27895.184} C_VEL
LIN {X 0,Y 166.806,Z 344.612,A -85,B 0,C 180,E1 -27899.397,E2 -27899.397} C_VEL
LIN {X 0,Y 166.785,Z 344.594,A -85,B 0,C 180,E1 -27903.009,E2 -27903.009} C_VEL
LIN {X 0,Y 167.029,Z 345.564,A -85,B 0,C 180,E1 -27905.493,E2 -27905.493} C_VEL
LIN {X 0,Y 167.689,Z 347.484,A -85,B 0,C 180,E1 -27908.587,E2 -27908.587} C_VEL
LIN {X 0,Y 168.905,Z 351.087,A -85,B 0,C 180,E1 -27912.163,E2 -27912.163} C_VEL
LIN {X 0,Y 170.554,Z 356.156,A -85,B 0,C 180,E1 -27915.626,E2 -27915.626} C_VEL
LIN {X 0,Y 171.456,Z 359.288,A -85,B 0,C 180,E1 -27917.231,E2 -27917.231} C_VEL
LIN {X 0,Y 167.233,Z 396.94,A -85,B 0,C 180,E1 -27918.138,E2 -27918.138} C_VEL
LIN {X 0,Y 164.293,Z 411.533,A -85,B 0,C 180,E1 -27918.677,E2 -27918.677} C_VEL
LIN {X 0,Y 160.289,Z 425.511,A -85,B 0,C 180,E1 -27919.492,E2 -27919.492} C_VEL
LIN {X 0,Y 155.584,Z 437.959,A -85,B 0,C 180,E1 -27920.394,E2 -27920.394} C_VEL
LIN {X 0,Y 149.351,Z 451.107,A -85,B 0,C 180,E1 -27921.662,E2 -27921.662} C_VEL
LIN {X 0,Y 142.685,Z 462.9,A -85,B 0,C 180,E1 -27923.293,E2 -27923.293} C_VEL
LIN {X 0,Y 134.332,Z 475.137,A -85,B 0,C 180,E1 -27925.512,E2 -27925.512} C_VEL
LIN {X 0,Y 126.904,Z 484.346,A -85,B 0,C 180,E1 -27927.614,E2 -27927.614} C_VEL
LIN {X 0,Y 118.405,Z 493.635,A -85,B 0,C 180,E1 -27930.609,E2 -27930.609} C_VEL
LIN {X 0,Y 108.813,Z 502.646,A -85,B 0,C 180,E1 -27934.562,E2 -27934.562} C_VEL
LIN {X 0,Y 99.889,Z 510.001,A -85,B 0,C 180,E1 -27939.289,E2 -27939.289} C_VEL
LIN {X 0,Y 93.057,Z 515.151,A -85,B 0,C 180,E1 -27944.152,E2 -27944.152} C_VEL
LIN {X 0,Y 84.604,Z 520.695,A -85,B 0,C 180,E1 -27951.462,E2 -27951.462} C_VEL
LIN {X 0,Y 79.449,Z 523.901,A -85,B 0,C 180,E1 -27957.942,E2 -27957.942} C_VEL
LIN {X 0,Y 74.24,Z 526.977,A -85,B 0,C 180,E1 -27967.747,E2 -27967.747} C_VEL
LIN {X 0,Y 71.114,Z 528.8,A -85,B 0,C 180,E1 -27978.598,E2 -27978.598} C_VEL
LIN {X 0,Y 70.138,Z 529.41,A -85,B 0,C 180,E1 -27989.998,E2 -27989.998} C_VEL
LIN {X 0,Y 71.048,Z 528.833,A -85,B 0,C 180,E1 -28001.408,E2 -28001.408} C_VEL
LIN {X 0,Y 74.183,Z 527.048,A -85,B 0,C 180,E1 -28012.267,E2 -28012.267} C_VEL
LIN {X 0,Y 79.413,Z 524.003,A -85,B 0,C 180,E1 -28022.07,E2 -28022.07} C_VEL
LIN {X 0,Y 86.511,Z 519.614,A -85,B 0,C 180,E1 -28030.532,E2 -28030.532} C_VEL
LIN {X 0,Y 95.177,Z 513.757,A -85,B 0,C 180,E1 -28037.593,E2 -28037.593} C_VEL
LIN {X 0,Y 103.579,Z 507.254,A -85,B 0,C 180,E1 -28042.866,E2 -28042.866} C_VEL
LIN {X 0,Y 112.812,Z 499.277,A -85,B 0,C 180,E1 -28047.245,E2 -28047.245} C_VEL
LIN {X 0,Y 122.594,Z 489.551,A -85,B 0,C 180,E1 -28050.952,E2 -28050.952} C_VEL
LIN {X 0,Y 131.272,Z 479.436,A -85,B 0,C 180,E1 -28053.731,E2 -28053.731} C_VEL
LIN {X 0,Y 138.759,Z 469.352,A -85,B 0,C 180,E1 -28055.735,E2 -28055.735} C_VEL
LIN {X 0,Y 146.244,Z 457.327,A -85,B 0,C 180,E1 -28057.677,E2 -28057.677} C_VEL
LIN {X 0,Y 153.173,Z 444.014,A -85,B 0,C 180,E1 -28059.2,E2 -28059.2} C_VEL
LIN {X 0,Y 159.034,Z 429.893,A -85,B 0,C 180,E1 -28060.357,E2 -28060.357} C_VEL
LIN {X 0,Y 163.55,Z 415.632,A -85,B 0,C 180,E1 -28061.214,E2 -28061.214} C_VEL
LIN {X 0,Y 166.714,Z 401.588,A -85,B 0,C 180,E1 -28061.845,E2 -28061.845} C_VEL
LIN {X 0,Y 168.985,Z 385.496,A -85,B 0,C 180,E1 -28062.259,E2 -28062.259} C_VEL
LIN {X 0,Y 171.723,Z 359.479,A -85,B 0,C 180,E1 -28062.912,E2 -28062.912} C_VEL
LIN {X 0,Y 170.335,Z 354.879,A -85,B 0,C 180,E1 -28065.466,E2 -28065.466} C_VEL
LIN {X 0,Y 168.966,Z 350.519,A -85,B 0,C 180,E1 -28068.605,E2 -28068.605} C_VEL
LIN {X 0,Y 167.76,Z 347.051,A -85,B 0,C 180,E1 -28072.477,E2 -28072.477} C_VEL
LIN {X 0,Y 167.141,Z 345.077,A -85,B 0,C 180,E1 -28076.383,E2 -28076.383} C_VEL
LIN {X 0,Y 167.08,Z 344.741,A -85,B 0,C 180,E1 -28080,E2 -28080} C_VEL
LIN {X 0,Y 167.573,Z 346.601,A -85,B 0,C 180,E1 -28084.209,E2 -28084.209} C_VEL
LIN {X 0,Y 168.024,Z 348.145,A -85,B 0,C 180,E1 -28086.153,E2 -28086.153} C_VEL
LIN {X 0,Y 169.023,Z 351.243,A -85,B 0,C 180,E1 -28089.136,E2 -28089.136} C_VEL
LIN {X 0,Y 170.12,Z 354.632,A -85,B 0,C 180,E1 -28091.618,E2 -28091.618} C_VEL
LIN {X 0,Y 171.677,Z 359.862,A -85,B 0,C 180,E1 -28094.521,E2 -28094.521} C_VEL
LIN {X 0,Y 167.199,Z 399.273,A -85,B 0,C 180,E1 -28095.49,E2 -28095.49} C_VEL
LIN {X 0,Y 164.127,Z 414.148,A -85,B 0,C 180,E1 -28095.97,E2 -28095.97} C_VEL
LIN {X 0,Y 160.004,Z 428.172,A -85,B 0,C 180,E1 -28096.653,E2 -28096.653} C_VEL
LIN {X 0,Y 154.81,Z 441.706,A -85,B 0,C 180,E1 -28097.576,E2 -28097.576} C_VEL
LIN {X 0,Y 148.424,Z 454.89,A -85,B 0,C 180,E1 -28098.74,E2 -28098.74} C_VEL
LIN {X 0,Y 141.112,Z 467.43,A -85,B 0,C 180,E1 -28100.31,E2 -28100.31} C_VEL
LIN {X 0,Y 132.951,Z 479.227,A -85,B 0,C 180,E1 -28102.325,E2 -28102.325} C_VEL
LIN {X 0,Y 123.911,Z 490.267,A -85,B 0,C 180,E1 -28104.844,E2 -28104.844} C_VEL
LIN {X 0,Y 115.23,Z 499.536,A -85,B 0,C 180,E1 -28107.83,E2 -28107.83} C_VEL
LIN {X 0,Y 105.754,Z 508.444,A -85,B 0,C 180,E1 -28111.928,E2 -28111.928} C_VEL
LIN {X 0,Y 96.766,Z 515.976,A -85,B 0,C 180,E1 -28116.977,E2 -28116.977} C_VEL
LIN {X 0,Y 87.56,Z 522.782,A -85,B 0,C 180,E1 -28123.752,E2 -28123.752} C_VEL
LIN {X 0,Y 79.932,Z 528.056,A -85,B 0,C 180,E1 -28132.017,E2 -28132.017} C_VEL
LIN {X 0,Y 74.176,Z 531.932,A -85,B 0,C 180,E1 -28141.726,E2 -28141.726} C_VEL
LIN {X 0,Y 70.69,Z 534.496,A -85,B 0,C 180,E1 -28152.649,E2 -28152.649} C_VEL
LIN {X 0,Y 69.691,Z 535.804,A -85,B 0,C 180,E1 -28164.214,E2 -28164.214} C_VEL
LIN {X 0,Y 69.948,Z 535.983,A -85,B 0,C 180,E1 -28170.002,E2 -28170.002} C_VEL
LIN {X 0,Y 69.925,Z 535.285,A -85,B 0,C 180,E1 -28181.598,E2 -28181.598} C_VEL
LIN {X 0,Y 72.111,Z 533.321,A -85,B 0,C 180,E1 -28192.947,E2 -28192.947} C_VEL
LIN {X 0,Y 76.815,Z 530.088,A -85,B 0,C 180,E1 -28203.297,E2 -28203.297} C_VEL
LIN {X 0,Y 83.529,Z 525.5,A -85,B 0,C 180,E1 -28212.309,E2 -28212.309} C_VEL
LIN {X 0,Y 91.987,Z 519.443,A -85,B 0,C 180,E1 -28219.821,E2 -28219.821} C_VEL
LIN {X 0,Y 100.488,Z 512.777,A -85,B 0,C 180,E1 -28225.265,E2 -28225.265} C_VEL
LIN {X 0,Y 109.652,Z 504.664,A -85,B 0,C 180,E1 -28229.915,E2 -28229.915} C_VEL
LIN {X 0,Y 118.101,Z 496.346,A -85,B 0,C 180,E1 -28233.206,E2 -28233.206} C_VEL
LIN {X 0,Y 126.894,Z 486.49,A -85,B 0,C 180,E1 -28236.044,E2 -28236.044} C_VEL
LIN {X 0,Y 135.983,Z 474.66,A -85,B 0,C 180,E1 -28238.481,E2 -28238.481} C_VEL
LIN {X 0,Y 141.066,Z 467.061,A -85,B 0,C 180,E1 -28239.715,E2 -28239.715} C_VEL
LIN {X 0,Y 143.816,Z 462.306,A -85,B 0,C 180,E1 -28240.586,E2 -28240.586} C_VEL
LIN {X 0,Y 147.22,Z 454.421,A -85,B 0,C 180,E1 -28242.541,E2 -28242.541} C_VEL
LIN {X 0,Y 150.371,Z 446.305,A -85,B 0,C 180,E1 -28244.338,E2 -28244.338} C_VEL
LIN {X 0,Y 152.578,Z 441.046,A -85,B 0,C 180,E1 -28244.983,E2 -28244.983} C_VEL
LIN {X 0,Y 157.695,Z 427.981,A -85,B 0,C 180,E1 -28245.774,E2 -28245.774} C_VEL
LIN {X 0,Y 162.159,Z 413.052,A -85,B 0,C 180,E1 -28246.414,E2 -28246.414} C_VEL
LIN {X 0,Y 165.256,Z 397.561,A -85,B 0,C 180,E1 -28246.892,E2 -28246.892} C_VEL
LIN {X 0,Y 169.16,Z 363.43,A -85,B 0,C 180,E1 -28247.707,E2 -28247.707} C_VEL
LIN {X 0,Y 167.761,Z 358.372,A -85,B 0,C 180,E1 -28250.962,E2 -28250.962} C_VEL
LIN {X 0,Y 166.88,Z 355.401,A -85,B 0,C 180,E1 -28253.653,E2 -28253.653} C_VEL
LIN {X 0,Y 166.393,Z 353.563,A -85,B 0,C 180,E1 -28255.762,E2 -28255.762} C_VEL
LIN {X 0,Y 165.938,Z 351.683,A -85,B 0,C 180,E1 -28259.394,E2 -28259.394} C_VEL
LIN {X 0,Y 165.918,Z 351.663,A -85,B 0,C 180,E1 -28263.024,E2 -28263.024} C_VEL
LIN {X 0,Y 166.239,Z 353.024,A -85,B 0,C 180,E1 -28266.067,E2 -28266.067} C_VEL
LIN {X 0,Y 166.678,Z 354.482,A -85,B 0,C 180,E1 -28268.182,E2 -28268.182} C_VEL
LIN {X 0,Y 167.694,Z 357.799,A -85,B 0,C 180,E1 -28271.473,E2 -28271.473} C_VEL
LIN {X 0,Y 169.233,Z 363.146,A -85,B 0,C 180,E1 -28275.023,E2 -28275.023} C_VEL
LIN {X 0,Y 165.373,Z 396.671,A -85,B 0,C 180,E1 -28275.771,E2 -28275.771} C_VEL
LIN {X 0,Y 162.419,Z 411.246,A -85,B 0,C 180,E1 -28276.272,E2 -28276.272} C_VEL
LIN {X 0,Y 158.47,Z 424.924,A -85,B 0,C 180,E1 -28277.004,E2 -28277.004} C_VEL
LIN {X 0,Y 153.264,Z 438.425,A -85,B 0,C 180,E1 -28277.916,E2 -28277.916} C_VEL
LIN {X 0,Y 146.888,Z 451.529,A -85,B 0,C 180,E1 -28279.098,E2 -28279.098} C_VEL
LIN {X 0,Y 139.766,Z 463.704,A -85,B 0,C 180,E1 -28280.696,E2 -28280.696} C_VEL
LIN {X 0,Y 131.435,Z 475.511,A -85,B 0,C 180,E1 -28282.723,E2 -28282.723} C_VEL
LIN {X 0,Y 123.778,Z 484.711,A -85,B 0,C 180,E1 -28284.705,E2 -28284.705} C_VEL
LIN {X 0,Y 114.962,Z 493.99,A -85,B 0,C 180,E1 -28287.571,E2 -28287.571} C_VEL
LIN {X 0,Y 104.954,Z 502.991,A -85,B 0,C 180,E1 -28291.374,E2 -28291.374} C_VEL
LIN {X 0,Y 95.14,Z 510.644,A -85,B 0,C 180,E1 -28296.226,E2 -28296.226} C_VEL
LIN {X 0,Y 88.26,Z 515.489,A -85,B 0,C 180,E1 -28300.845,E2 -28300.845} C_VEL
LIN {X 0,Y 79.183,Z 521.03,A -85,B 0,C 180,E1 -28308.264,E2 -28308.264} C_VEL
LIN {X 0,Y 73.53,Z 524.235,A -85,B 0,C 180,E1 -28315.005,E2 -28315.005} C_VEL
LIN {X 0,Y 67.727,Z 527.31,A -85,B 0,C 180,E1 -28325.474,E2 -28325.474} C_VEL
LIN {X 0,Y 64.175,Z 529.133,A -85,B 0,C 180,E1 -28337.346,E2 -28337.346} C_VEL
LIN {X 0,Y 63.058,Z 529.742,A -85,B 0,C 180,E1 -28349.998,E2 -28349.998} C_VEL
LIN {X 0,Y 64.101,Z 529.166,A -85,B 0,C 180,E1 -28362.664,E2 -28362.664} C_VEL
LIN {X 0,Y 67.654,Z 527.381,A -85,B 0,C 180,E1 -28374.55,E2 -28374.55} C_VEL
LIN {X 0,Y 73.497,Z 524.335,A -85,B 0,C 180,E1 -28385.008,E2 -28385.008} C_VEL
LIN {X 0,Y 81.258,Z 519.947,A -85,B 0,C 180,E1 -28393.779,E2 -28393.779} C_VEL
LIN {X 0,Y 88.16,Z 515.673,A -85,B 0,C 180,E1 -28399.226,E2 -28399.226} C_VEL
LIN {X 0,Y 95.511,Z 510.563,A -85,B 0,C 180,E1 -28404.035,E2 -28404.035} C_VEL
LIN {X 0,Y 104.881,Z 503.254,A -85,B 0,C 180,E1 -28408.686,E2 -28408.686} C_VEL
LIN {X 0,Y 114.917,Z 494.314,A -85,B 0,C 180,E1 -28412.467,E2 -28412.467} C_VEL
LIN {X 0,Y 123.741,Z 485.084,A -85,B 0,C 180,E1 -28415.327,E2 -28415.327} C_VEL
LIN {X 0,Y 132.88,Z 473.978,A -85,B 0,C 180,E1 -28417.749,E2 -28417.749} C_VEL
LIN {X 0,Y 139.881,Z 463.944,A -85,B 0,C 180,E1 -28419.408,E2 -28419.408} C_VEL
LIN {X 0,Y 146.849,Z 452.154,A -85,B 0,C 180,E1 -28420.94,E2 -28420.94} C_VEL
LIN {X 0,Y 153.219,Z 439.205,A -85,B 0,C 180,E1 -28422.129,E2 -28422.129} C_VEL
LIN {X 0,Y 158.388,Z 425.913,A -85,B 0,C 180,E1 -28423.086,E2 -28423.086} C_VEL
LIN {X 0,Y 162.696,Z 411.319,A -85,B 0,C 180,E1 -28423.841,E2 -28423.841} C_VEL
LIN {X 0,Y 165.642,Z 396.862,A -85,B 0,C 180,E1 -28424.335,E2 -28424.335} C_VEL
LIN {X 0,Y 169.537,Z 363.463,A -85,B 0,C 180,E1 -28425.079,E2 -28425.079} C_VEL
LIN {X 0,Y 168.046,Z 358.202,A -85,B 0,C 180,E1 -28428.541,E2 -28428.541} C_VEL
LIN {X 0,Y 167.099,Z 355.138,A -85,B 0,C 180,E1 -28431.499,E2 -28431.499} C_VEL
LIN {X 0,Y 166.619,Z 353.555,A -85,B 0,C 180,E1 -28433.643,E2 -28433.643} C_VEL
LIN {X 0,Y 166.229,Z 351.997,A -85,B 0,C 180,E1 -28436.97,E2 -28436.97} C_VEL
LIN {X 0,Y 166.235,Z 352.015,A -85,B 0,C 180,E1 -28440.605,E2 -28440.605} C_VEL
LIN {X 0,Y 166.788,Z 354.082,A -85,B 0,C 180,E1 -28444.682,E2 -28444.682} C_VEL
LIN {X 0,Y 167.781,Z 357.814,A -85,B 0,C 180,E1 -28448.338,E2 -28448.338} C_VEL
LIN {X 0,Y 168.774,Z 361.301,A -85,B 0,C 180,E1 -28450.866,E2 -28450.866} C_VEL
LIN {X 0,Y 169.425,Z 363.678,A -85,B 0,C 180,E1 -28452.274,E2 -28452.274} C_VEL
LIN {X 0,Y 165.415,Z 398.559,A -85,B 0,C 180,E1 -28453.122,E2 -28453.122} C_VEL
LIN {X 0,Y 162.299,Z 413.558,A -85,B 0,C 180,E1 -28453.554,E2 -28453.554} C_VEL
LIN {X 0,Y 158.116,Z 427.648,A -85,B 0,C 180,E1 -28454.187,E2 -28454.187} C_VEL
LIN {X 0,Y 152.808,Z 441.247,A -85,B 0,C 180,E1 -28455.025,E2 -28455.025} C_VEL
LIN {X 0,Y 146.285,Z 454.472,A -85,B 0,C 180,E1 -28456.089,E2 -28456.089} C_VEL
LIN {X 0,Y 139.144,Z 466.515,A -85,B 0,C 180,E1 -28457.465,E2 -28457.465} C_VEL
LIN {X 0,Y 130.405,Z 478.857,A -85,B 0,C 180,E1 -28459.42,E2 -28459.42} C_VEL
LIN {X 0,Y 121.082,Z 489.91,A -85,B 0,C 180,E1 -28461.774,E2 -28461.774} C_VEL
LIN {X 0,Y 112.067,Z 499.187,A -85,B 0,C 180,E1 -28464.592,E2 -28464.592} C_VEL
LIN {X 0,Y 101.766,Z 508.398,A -85,B 0,C 180,E1 -28468.666,E2 -28468.666} C_VEL
LIN {X 0,Y 92.612,Z 515.635,A -85,B 0,C 180,E1 -28473.415,E2 -28473.415} C_VEL
LIN {X 0,Y 82.76,Z 522.444,A -85,B 0,C 180,E1 -28480.161,E2 -28480.161} C_VEL
LIN {X 0,Y 74.396,Z 527.719,A -85,B 0,C 180,E1 -28488.606,E2 -28488.606} C_VEL
LIN {X 0,Y 67.93,Z 531.595,A -85,B 0,C 180,E1 -28498.852,E2 -28498.852} C_VEL
LIN {X 0,Y 63.896,Z 534.161,A -85,B 0,C 180,E1 -28510.736,E2 -28510.736} C_VEL
LIN {X 0,Y 62.588,Z 535.469,A -85,B 0,C 180,E1 -28523.555,E2 -28523.555} C_VEL
LIN {X 0,Y 62.841,Z 535.65,A -85,B 0,C 180,E1 -28530.002,E2 -28530.002} C_VEL
LIN {X 0,Y 62.923,Z 534.949,A -85,B 0,C 180,E1 -28542.91,E2 -28542.91} C_VEL
LIN {X 0,Y 65.572,Z 532.984,A -85,B 0,C 180,E1 -28555.389,E2 -28555.389} C_VEL
LIN {X 0,Y 70.908,Z 529.749,A -85,B 0,C 180,E1 -28566.492,E2 -28566.492} C_VEL
LIN {X 0,Y 78.358,Z 525.16,A -85,B 0,C 180,E1 -28575.853,E2 -28575.853} C_VEL
LIN {X 0,Y 87.534,Z 519.102,A -85,B 0,C 180,E1 -28583.409,E2 -28583.409} C_VEL
LIN {X 0,Y 97.911,Z 511.397,A -85,B 0,C 180,E1 -28589.47,E2 -28589.47} C_VEL
LIN {X 0,Y 107.671,Z 503.055,A -85,B 0,C 180,E1 -28593.833,E2 -28593.833} C_VEL
LIN {X 0,Y 118.037,Z 492.913,A -85,B 0,C 180,E1 -28597.352,E2 -28597.352} C_VEL
LIN {X 0,Y 127.28,Z 482.452,A -85,B 0,C 180,E1 -28599.834,E2 -28599.834} C_VEL
LIN {X 0,Y 135.59,Z 471.362,A -85,B 0,C 180,E1 -28601.828,E2 -28601.828} C_VEL
LIN {X 0,Y 143.047,Z 459.698,A -85,B 0,C 180,E1 -28603.346,E2 -28603.346} C_VEL
LIN {X 0,Y 150.344,Z 445.927,A -85,B 0,C 180,E1 -28604.611,E2 -28604.611} C_VEL
LIN {X 0,Y 152.578,Z 441.046,A -85,B 0,C 180,E1 -28604.983,E2 -28604.983} C_VEL
LIN {X 0,Y 154.682,Z 435.754,A -85,B 0,C 180,E1 -28605.582,E2 -28605.582} C_VEL
LIN {X 0,Y 157.147,Z 427.061,A -85,B 0,C 180,E1 -28607.105,E2 -28607.105} C_VEL
LIN {X 0,Y 159.207,Z 418.151,A -85,B 0,C 180,E1 -28608.486,E2 -28608.486} C_VEL
LIN {X 0,Y 160.597,Z 412.525,A -85,B 0,C 180,E1 -28608.874,E2 -28608.874} C_VEL
LIN {X 0,Y 163.519,Z 398.277,A -85,B 0,C 180,E1 -28609.284,E2 -28609.284} C_VEL
LIN {X 0,Y 167.163,Z 367.623,A -85,B 0,C 180,E1 -28609.947,E2 -28609.947} C_VEL
LIN {X 0,Y 166.18,Z 363.603,A -85,B 0,C 180,E1 -28612.864,E2 -28612.864} C_VEL
LIN {X 0,Y 165.453,Z 360.556,A -85,B 0,C 180,E1 -28616.042,E2 -28616.042} C_VEL
LIN {X 0,Y 165.041,Z 358.59,A -85,B 0,C 180,E1 -28620,E2 -28620} C_VEL
LIN {X 0,Y 165.094,Z 358.863,A -85,B 0,C 180,E1 -28623.639,E2 -28623.639} C_VEL
LIN {X 0,Y 165.588,Z 361.038,A -85,B 0,C 180,E1 -28627.316,E2 -28627.316} C_VEL
LIN {X 0,Y 166.5,Z 364.508,A -85,B 0,C 180,E1 -28630.757,E2 -28630.757} C_VEL
LIN {X 0,Y 167.213,Z 367.39,A -85,B 0,C 180,E1 -28632.747,E2 -28632.747} C_VEL
LIN {X 0,Y 163.637,Z 397.326,A -85,B 0,C 180,E1 -28633.383,E2 -28633.383} C_VEL
LIN {X 0,Y 160.585,Z 411.883,A -85,B 0,C 180,E1 -28633.846,E2 -28633.846} C_VEL
LIN {X 0,Y 156.552,Z 425.458,A -85,B 0,C 180,E1 -28634.535,E2 -28634.535} C_VEL
LIN {X 0,Y 151.239,Z 438.891,A -85,B 0,C 180,E1 -28635.368,E2 -28635.368} C_VEL
LIN {X 0,Y 144.731,Z 451.951,A -85,B 0,C 180,E1 -28636.454,E2 -28636.454} C_VEL
LIN {X 0,Y 137.897,Z 463.376,A -85,B 0,C 180,E1 -28637.806,E2 -28637.806} C_VEL
LIN {X 0,Y 130.454,Z 473.888,A -85,B 0,C 180,E1 -28639.475,E2 -28639.475} C_VEL
LIN {X 0,Y 120.99,Z 485.074,A -85,B 0,C 180,E1 -28641.658,E2 -28641.658} C_VEL
LIN {X 0,Y 111.859,Z 494.345,A -85,B 0,C 180,E1 -28644.351,E2 -28644.351} C_VEL
LIN {X 0,Y 101.437,Z 503.337,A -85,B 0,C 180,E1 -28647.946,E2 -28647.946} C_VEL
LIN {X 0,Y 90.722,Z 511.251,A -85,B 0,C 180,E1 -28652.839,E2 -28652.839} C_VEL
LIN {X 0,Y 81.24,Z 517.384,A -85,B 0,C 180,E1 -28658.867,E2 -28658.867} C_VEL
LIN {X 0,Y 71.81,Z 522.538,A -85,B 0,C 180,E1 -28666.756,E2 -28666.756} C_VEL
LIN {X 0,Y 64.296,Z 526.269,A -85,B 0,C 180,E1 -28676.868,E2 -28676.868} C_VEL
LIN {X 0,Y 58.971,Z 528.708,A -85,B 0,C 180,E1 -28689.049,E2 -28689.049} C_VEL
LIN {X 0,Y 56.295,Z 529.919,A -85,B 0,C 180,E1 -28702.826,E2 -28702.826} C_VEL
LIN {X 0,Y 55.978,Z 530.075,A -85,B 0,C 180,E1 -28709.997,E2 -28709.997} C_VEL
LIN {X 0,Y 57.21,Z 529.498,A -85,B 0,C 180,E1 -28724.22,E2 -28724.22} C_VEL
LIN {X 0,Y 61.266,Z 527.713,A -85,B 0,C 180,E1 -28737.31,E2 -28737.31} C_VEL
LIN {X 0,Y 67.805,Z 524.668,A -85,B 0,C 180,E1 -28748.451,E2 -28748.451} C_VEL
LIN {X 0,Y 73.97,Z 521.5,A -85,B 0,C 180,E1 -28755.442,E2 -28755.442} C_VEL
LIN {X 0,Y 83.686,Z 516.008,A -85,B 0,C 180,E1 -28762.918,E2 -28762.918} C_VEL
LIN {X 0,Y 91.517,Z 510.9,A -85,B 0,C 180,E1 -28767.64,E2 -28767.64} C_VEL
LIN {X 0,Y 101.379,Z 503.594,A -85,B 0,C 180,E1 -28772.11,E2 -28772.11} C_VEL
LIN {X 0,Y 111.809,Z 494.664,A -85,B 0,C 180,E1 -28775.698,E2 -28775.698} C_VEL
LIN {X 0,Y 120.956,Z 485.439,A -85,B 0,C 180,E1 -28778.376,E2 -28778.376} C_VEL
LIN {X 0,Y 130.368,Z 474.351,A -85,B 0,C 180,E1 -28780.626,E2 -28780.626} C_VEL
LIN {X 0,Y 137.196,Z 464.845,A -85,B 0,C 180,E1 -28782.1,E2 -28782.1} C_VEL
LIN {X 0,Y 143.887,Z 453.983,A -85,B 0,C 180,E1 -28783.441,E2 -28783.441} C_VEL
LIN {X 0,Y 150.388,Z 441.418,A -85,B 0,C 180,E1 -28784.542,E2 -28784.542} C_VEL
LIN {X 0,Y 156.067,Z 427.561,A -85,B 0,C 180,E1 -28785.501,E2 -28785.501} C_VEL
LIN {X 0,Y 160.541,Z 413.193,A -85,B 0,C 180,E1 -28786.206,E2 -28786.206} C_VEL
LIN {X 0,Y 163.7,Z 398.662,A -85,B 0,C 180,E1 -28786.702,E2 -28786.702} C_VEL
LIN {X 0,Y 166.872,Z 373.533,A -85,B 0,C 180,E1 -28787.218,E2 -28787.218} C_VEL
LIN {X 0,Y 167.511,Z 367.579,A -85,B 0,C 180,E1 -28787.399,E2 -28787.399} C_VEL
LIN {X 0,Y 166.536,Z 363.631,A -85,B 0,C 180,E1 -28790.281,E2 -28790.281} C_VEL
LIN {X 0,Y 165.746,Z 360.711,A -85,B 0,C 180,E1 -28793.609,E2 -28793.609} C_VEL
LIN {X 0,Y 165.363,Z 359.061,A -85,B 0,C 180,E1 -28796.954,E2 -28796.954} C_VEL
LIN {X 0,Y 165.35,Z 359.006,A -85,B 0,C 180,E1 -28800.304,E2 -28800.304} C_VEL
LIN {X 0,Y 165.752,Z 360.802,A -85,B 0,C 180,E1 -28803.95,E2 -28803.95} C_VEL
LIN {X 0,Y 166.604,Z 364.521,A -85,B 0,C 180,E1 -28807.616,E2 -28807.616} C_VEL
LIN {X 0,Y 167.443,Z 367.867,A -85,B 0,C 180,E1 -28810.04,E2 -28810.04} C_VEL
LIN {X 0,Y 163.785,Z 398.53,A -85,B 0,C 180,E1 -28810.706,E2 -28810.706} C_VEL
LIN {X 0,Y 160.534,Z 413.82,A -85,B 0,C 180,E1 -28811.121,E2 -28811.121} C_VEL
LIN {X 0,Y 156.106,Z 428.258,A -85,B 0,C 180,E1 -28811.716,E2 -28811.716} C_VEL
LIN {X 0,Y 151.118,Z 440.789,A -85,B 0,C 180,E1 -28812.416,E2 -28812.416} C_VEL
LIN {X 0,Y 144.473,Z 454.056,A -85,B 0,C 180,E1 -28813.373,E2 -28813.373} C_VEL
LIN {X 0,Y 137.01,Z 466.361,A -85,B 0,C 180,E1 -28814.652,E2 -28814.652} C_VEL
LIN {X 0,Y 128.212,Z 478.487,A -85,B 0,C 180,E1 -28816.415,E2 -28816.415} C_VEL
LIN {X 0,Y 118.621,Z 489.554,A -85,B 0,C 180,E1 -28818.572,E2 -28818.572} C_VEL
LIN {X 0,Y 109.286,Z 498.839,A -85,B 0,C 180,E1 -28821.183,E2 -28821.183} C_VEL
LIN {X 0,Y 98.756,Z 507.87,A -85,B 0,C 180,E1 -28824.898,E2 -28824.898} C_VEL
LIN {X 0,Y 88.838,Z 515.293,A -85,B 0,C 180,E1 -28829.521,E2 -28829.521} C_VEL
LIN {X 0,Y 78.319,Z 522.106,A -85,B 0,C 180,E1 -28836.141,E2 -28836.141} C_VEL
LIN {X 0,Y 69.167,Z 527.382,A -85,B 0,C 180,E1 -28844.666,E2 -28844.666} C_VEL
LIN {X 0,Y 61.888,Z 531.258,A -85,B 0,C 180,E1 -28855.407,E2 -28855.407} C_VEL
LIN {X 0,Y 57.18,Z 533.825,A -85,B 0,C 180,E1 -28868.366,E2 -28868.366} C_VEL
LIN {X 0,Y 55.513,Z 535.135,A -85,B 0,C 180,E1 -28882.73,E2 -28882.73} C_VEL
LIN {X 0,Y 55.718,Z 535.316,A -85,B 0,C 180,E1 -28890.003,E2 -28890.003} C_VEL
LIN {X 0,Y 55.978,Z 534.613,A -85,B 0,C 180,E1 -28904.545,E2 -28904.545} C_VEL
LIN {X 0,Y 59.181,Z 532.648,A -85,B 0,C 180,E1 -28918.363,E2 -28918.363} C_VEL
LIN {X 0,Y 65.249,Z 529.41,A -85,B 0,C 180,E1 -28930.263,E2 -28930.263} C_VEL
LIN {X 0,Y 73.538,Z 524.821,A -85,B 0,C 180,E1 -28939.869,E2 -28939.869} C_VEL
LIN {X 0,Y 83.459,Z 518.761,A -85,B 0,C 180,E1 -28947.364,E2 -28947.364} C_VEL
LIN {X 0,Y 94.446,Z 511.048,A -85,B 0,C 180,E1 -28953.248,E2 -28953.248} C_VEL
LIN {X 0,Y 104.711,Z 502.703,A -85,B 0,C 180,E1 -28957.351,E2 -28957.351} C_VEL
LIN {X 0,Y 115.463,Z 492.548,A -85,B 0,C 180,E1 -28960.641,E2 -28960.641} C_VEL
LIN {X 0,Y 124.993,Z 482.074,A -85,B 0,C 180,E1 -28962.914,E2 -28962.914} C_VEL
LIN {X 0,Y 133.725,Z 470.699,A -85,B 0,C 180,E1 -28964.766,E2 -28964.766} C_VEL
LIN {X 0,Y 141.171,Z 459.275,A -85,B 0,C 180,E1 -28966.116,E2 -28966.116} C_VEL
LIN {X 0,Y 148.614,Z 445.458,A -85,B 0,C 180,E1 -28967.256,E2 -28967.256} C_VEL
LIN {X 0,Y 154.427,Z 431.968,A -85,B 0,C 180,E1 -28968.089,E2 -28968.089} C_VEL
LIN {X 0,Y 159.204,Z 417.608,A -85,B 0,C 180,E1 -28968.708,E2 -28968.708} C_VEL
LIN {X 0,Y 160.597,Z 412.525,A -85,B 0,C 180,E1 -28968.874,E2 -28968.874} C_VEL
LIN {X 0,Y 161.82,Z 406.843,A -85,B 0,C 180,E1 -28969.238,E2 -28969.238} C_VEL
LIN {X 0,Y 162.944,Z 397.627,A -85,B 0,C 180,E1 -28970.471,E2 -28970.471} C_VEL
LIN {X 0,Y 163.638,Z 388.335,A -85,B 0,C 180,E1 -28971.715,E2 -28971.715} C_VEL
LIN {X 0,Y 164.18,Z 382.521,A -85,B 0,C 180,E1 -28972.082,E2 -28972.082} C_VEL
LIN {X 0,Y 165.399,Z 371.95,A -85,B 0,C 180,E1 -28972.288,E2 -28972.288} C_VEL
LIN {X 0,Y 164.708,Z 368.786,A -85,B 0,C 180,E1 -28975.105,E2 -28975.105} C_VEL
LIN {X 0,Y 164.373,Z 367.042,A -85,B 0,C 180,E1 -28977.243,E2 -28977.243} C_VEL
LIN {X 0,Y 164.172,Z 365.669,A -85,B 0,C 180,E1 -28980,E2 -28980} C_VEL
LIN {X 0,Y 164.203,Z 365.876,A -85,B 0,C 180,E1 -28983.357,E2 -28983.357} C_VEL
LIN {X 0,Y 164.604,Z 368.03,A -85,B 0,C 180,E1 -28986.897,E2 -28986.897} C_VEL
LIN {X 0,Y 165.288,Z 371.025,A -85,B 0,C 180,E1 -28989.862,E2 -28989.862} C_VEL
LIN {X 0,Y 165.449,Z 371.725,A -85,B 0,C 180,E1 -28990.413,E2 -28990.413} C_VEL
LIN {X 0,Y 162.146,Z 398.256,A -85,B 0,C 180,E1 -28990.967,E2 -28990.967} C_VEL
LIN {X 0,Y 159.038,Z 412.546,A -85,B 0,C 180,E1 -28991.372,E2 -28991.372} C_VEL
LIN {X 0,Y 154.511,Z 427.116,A -85,B 0,C 180,E1 -28992.057,E2 -28992.057} C_VEL
LIN {X 0,Y 148.705,Z 441.11,A -85,B 0,C 180,E1 -28992.898,E2 -28992.898} C_VEL
LIN {X 0,Y 142.06,Z 453.793,A -85,B 0,C 180,E1 -28993.858,E2 -28993.858} C_VEL
LIN {X 0,Y 135.021,Z 465.044,A -85,B 0,C 180,E1 -28995.149,E2 -28995.149} C_VEL
LIN {X 0,Y 126.639,Z 476.257,A -85,B 0,C 180,E1 -28996.8,E2 -28996.8} C_VEL
LIN {X 0,Y 116.976,Z 487.058,A -85,B 0,C 180,E1 -28998.866,E2 -28998.866} C_VEL
LIN {X 0,Y 107.565,Z 496.072,A -85,B 0,C 180,E1 -29001.399,E2 -29001.399} C_VEL
LIN {X 0,Y 96.799,Z 504.792,A -85,B 0,C 180,E1 -29004.828,E2 -29004.828} C_VEL
LIN {X 0,Y 86.48,Z 511.958,A -85,B 0,C 180,E1 -29009.184,E2 -29009.184} C_VEL
LIN {X 0,Y 76.992,Z 517.719,A -85,B 0,C 180,E1 -29014.758,E2 -29014.758} C_VEL
LIN {X 0,Y 66.808,Z 522.873,A -85,B 0,C 180,E1 -29022.574,E2 -29022.574} C_VEL
LIN {X 0,Y 58.48,Z 526.602,A -85,B 0,C 180,E1 -29033.064,E2 -29033.064} C_VEL
LIN {X 0,Y 52.418,Z 529.04,A -85,B 0,C 180,E1 -29046.28,E2 -29046.28} C_VEL
LIN {X 0,Y 49.278,Z 530.252,A -85,B 0,C 180,E1 -29061.798,E2 -29061.798} C_VEL
LIN {X 0,Y 49.262,Z 530.266,A -85,B 0,C 180,E1 -29078.199,E2 -29078.199} C_VEL
LIN {X 0,Y 52.354,Z 529.09,A -85,B 0,C 180,E1 -29093.745,E2 -29093.745} C_VEL
LIN {X 0,Y 58.44,Z 526.685,A -85,B 0,C 180,E1 -29106.96,E2 -29106.96} C_VEL
LIN {X 0,Y 66.759,Z 522.986,A -85,B 0,C 180,E1 -29117.465,E2 -29117.465} C_VEL
LIN {X 0,Y 76.926,Z 517.874,A -85,B 0,C 180,E1 -29125.306,E2 -29125.306} C_VEL
LIN {X 0,Y 87.923,Z 511.237,A -85,B 0,C 180,E1 -29131.55,E2 -29131.55} C_VEL
LIN {X 0,Y 98.256,Z 503.934,A -85,B 0,C 180,E1 -29135.774,E2 -29135.774} C_VEL
LIN {X 0,Y 109.079,Z 495.012,A -85,B 0,C 180,E1 -29139.099,E2 -29139.099} C_VEL
LIN {X 0,Y 118.53,Z 485.793,A -85,B 0,C 180,E1 -29141.56,E2 -29141.56} C_VEL
LIN {X 0,Y 128.197,Z 474.723,A -85,B 0,C 180,E1 -29143.607,E2 -29143.607} C_VEL
LIN {X 0,Y 135.321,Z 465.04,A -85,B 0,C 180,E1 -29144.981,E2 -29144.981} C_VEL
LIN {X 0,Y 142.854,Z 452.98,A -85,B 0,C 180,E1 -29146.315,E2 -29146.315} C_VEL
LIN {X 0,Y 149.483,Z 440.116,A -85,B 0,C 180,E1 -29147.3,E2 -29147.3} C_VEL
LIN {X 0,Y 154.871,Z 426.955,A -85,B 0,C 180,E1 -29148.089,E2 -29148.089} C_VEL
LIN {X 0,Y 159.319,Z 412.678,A -85,B 0,C 180,E1 -29148.724,E2 -29148.724} C_VEL
LIN {X 0,Y 162.422,Z 398.425,A -85,B 0,C 180,E1 -29149.159,E2 -29149.159} C_VEL
LIN {X 0,Y 165.769,Z 372.039,A -85,B 0,C 180,E1 -29149.661,E2 -29149.661} C_VEL
LIN {X 0,Y 165.155,Z 369.445,A -85,B 0,C 180,E1 -29151.988,E2 -29151.988} C_VEL
LIN {X 0,Y 164.713,Z 367.399,A -85,B 0,C 180,E1 -29154.49,E2 -29154.49} C_VEL
LIN {X 0,Y 164.471,Z 365.96,A -85,B 0,C 180,E1 -29157.551,E2 -29157.551} C_VEL
LIN {X 0,Y 164.492,Z 366.205,A -85,B 0,C 180,E1 -29160.612,E2 -29160.612} C_VEL
LIN {X 0,Y 164.801,Z 367.927,A -85,B 0,C 180,E1 -29163.667,E2 -29163.667} C_VEL
LIN {X 0,Y 165.448,Z 371.204,A -85,B 0,C 180,E1 -29166.861,E2 -29166.861} C_VEL
LIN {X 0,Y 165.693,Z 372.182,A -85,B 0,C 180,E1 -29167.705,E2 -29167.705} C_VEL
LIN {X 0,Y 162.506,Z 398.229,A -85,B 0,C 180,E1 -29168.249,E2 -29168.249} C_VEL
LIN {X 0,Y 159.195,Z 413.616,A -85,B 0,C 180,E1 -29168.624,E2 -29168.624} C_VEL
LIN {X 0,Y 154.819,Z 427.733,A -85,B 0,C 180,E1 -29169.138,E2 -29169.138} C_VEL
LIN {X 0,Y 149.744,Z 440.327,A -85,B 0,C 180,E1 -29169.746,E2 -29169.746} C_VEL
LIN {X 0,Y 142.996,Z 453.641,A -85,B 0,C 180,E1 -29170.601,E2 -29170.601} C_VEL
LIN {X 0,Y 135.553,Z 465.718,A -85,B 0,C 180,E1 -29171.695,E2 -29171.695} C_VEL
LIN {X 0,Y 126.363,Z 478.113,A -85,B 0,C 180,E1 -29173.276,E2 -29173.276} C_VEL
LIN {X 0,Y 116.548,Z 489.198,A -85,B 0,C 180,E1 -29175.25,E2 -29175.25} C_VEL
LIN {X 0,Y 106.903,Z 498.49,A -85,B 0,C 180,E1 -29177.595,E2 -29177.595} C_VEL
LIN {X 0,Y 95.816,Z 507.622,A -85,B 0,C 180,E1 -29181.04,E2 -29181.04} C_VEL
LIN {X 0,Y 85.522,Z 514.952,A -85,B 0,C 180,E1 -29185.323,E2 -29185.323} C_VEL
LIN {X 0,Y 74.302,Z 521.768,A -85,B 0,C 180,E1 -29191.653,E2 -29191.653} C_VEL
LIN {X 0,Y 64.31,Z 527.044,A -85,B 0,C 180,E1 -29200.1,E2 -29200.1} C_VEL
LIN {X 0,Y 56.117,Z 530.921,A -85,B 0,C 180,E1 -29211.234,E2 -29211.234} C_VEL
LIN {X 0,Y 50.571,Z 533.488,A -85,B 0,C 180,E1 -29225.364,E2 -29225.364} C_VEL
LIN {X 0,Y 48.446,Z 534.8,A -85,B 0,C 180,E1 -29241.662,E2 -29241.662} C_VEL
LIN {X 0,Y 48.617,Z 534.982,A -85,B 0,C 180,E1 -29250.003,E2 -29250.003} C_VEL
LIN {X 0,Y 49.072,Z 534.277,A -85,B 0,C 180,E1 -29266.648,E2 -29266.648} C_VEL
LIN {X 0,Y 52.99,Z 532.312,A -85,B 0,C 180,E1 -29282.043,E2 -29282.043} C_VEL
LIN {X 0,Y 59.935,Z 529.071,A -85,B 0,C 180,E1 -29294.716,E2 -29294.716} C_VEL
LIN {X 0,Y 69.119,Z 524.481,A -85,B 0,C 180,E1 -29304.436,E2 -29304.436} C_VEL
LIN {X 0,Y 79.821,Z 518.421,A -85,B 0,C 180,E1 -29311.701,E2 -29311.701} C_VEL
LIN {X 0,Y 91.425,Z 510.699,A -85,B 0,C 180,E1 -29317.29,E2 -29317.29} C_VEL
LIN {X 0,Y 102.161,Z 502.35,A -85,B 0,C 180,E1 -29321.071,E2 -29321.071} C_VEL
LIN {X 0,Y 113.291,Z 492.184,A -85,B 0,C 180,E1 -29324.061,E2 -29324.061} C_VEL
LIN {X 0,Y 123.081,Z 481.696,A -85,B 0,C 180,E1 -29326.1,E2 -29326.1} C_VEL
LIN {X 0,Y 131.292,Z 471.343,A -85,B 0,C 180,E1 -29327.637,E2 -29327.637} C_VEL
LIN {X 0,Y 139.628,Z 458.848,A -85,B 0,C 180,E1 -29328.965,E2 -29328.965} C_VEL
LIN {X 0,Y 146.361,Z 446.742,A -85,B 0,C 180,E1 -29329.858,E2 -29329.858} C_VEL
LIN {X 0,Y 152.693,Z 432.561,A -85,B 0,C 180,E1 -29330.646,E2 -29330.646} C_VEL
LIN {X 0,Y 157.615,Z 418.189,A -85,B 0,C 180,E1 -29331.215,E2 -29331.215} C_VEL
LIN {X 0,Y 161.139,Z 403.938,A -85,B 0,C 180,E1 -29331.598,E2 -29331.598} C_VEL
LIN {X 0,Y 163.513,Z 388.3,A -85,B 0,C 180,E1 -29331.971,E2 -29331.971} C_VEL
LIN {X 0,Y 164.18,Z 382.521,A -85,B 0,C 180,E1 -29332.082,E2 -29332.082} C_VEL
LIN {X 0,Y 164.345,Z 379.934,A -85,B 0,C 180,E1 -29332.425,E2 -29332.425} C_VEL
LIN {X 0,Y 164.269,Z 377.496,A -85,B 0,C 180,E1 -29333.318,E2 -29333.318} C_VEL
LIN {X 0,Y 164.02,Z 375.759,A -85,B 0,C 180,E1 -29334.572,E2 -29334.572} C_VEL
LIN {X 0,Y 163.599,Z 374.343,A -85,B 0,C 180,E1 -29336.666,E2 -29336.666} C_VEL
LIN {X 0,Y 163.345,Z 373.327,A -85,B 0,C 180,E1 -29338.802,E2 -29338.802} C_VEL
LIN {X 0,Y 163.303,Z 372.748,A -85,B 0,C 180,E1 -29340,E2 -29340} C_VEL
LIN {X 0,Y 163.319,Z 372.862,A -85,B 0,C 180,E1 -29343.073,E2 -29343.073} C_VEL
LIN {X 0,Y 163.633,Z 374.994,A -85,B 0,C 180,E1 -29346.474,E2 -29346.474} C_VEL
LIN {X 0,Y 163.93,Z 376.451,A -85,B 0,C 180,E1 -29348.068,E2 -29348.068} C_VEL
LIN {X 0,Y 161.112,Z 398.296,A -85,B 0,C 180,E1 -29348.484,E2 -29348.484} C_VEL
LIN {X 0,Y 158.094,Z 412.142,A -85,B 0,C 180,E1 -29348.825,E2 -29348.825} C_VEL
LIN {X 0,Y 153.619,Z 426.526,A -85,B 0,C 180,E1 -29349.433,E2 -29349.433} C_VEL
LIN {X 0,Y 148.124,Z 439.821,A -85,B 0,C 180,E1 -29350.094,E2 -29350.094} C_VEL
LIN {X 0,Y 141.38,Z 452.794,A -85,B 0,C 180,E1 -29350.954,E2 -29350.954} C_VEL
LIN {X 0,Y 135.002,Z 463.055,A -85,B 0,C 180,E1 -29351.923,E2 -29351.923} C_VEL
LIN {X 0,Y 126.44,Z 474.654,A -85,B 0,C 180,E1 -29353.413,E2 -29353.413} C_VEL
LIN {X 0,Y 116.512,Z 485.798,A -85,B 0,C 180,E1 -29355.176,E2 -29355.176} C_VEL
LIN {X 0,Y 106.794,Z 495.055,A -85,B 0,C 180,E1 -29357.401,E2 -29357.401} C_VEL
LIN {X 0,Y 95.619,Z 504.025,A -85,B 0,C 180,E1 -29360.424,E2 -29360.424} C_VEL
LIN {X 0,Y 84.806,Z 511.365,A -85,B 0,C 180,E1 -29364.272,E2 -29364.272} C_VEL
LIN {X 0,Y 73.183,Z 518.055,A -85,B 0,C 180,E1 -29370.195,E2 -29370.195} C_VEL
LIN {X 0,Y 62.218,Z 523.208,A -85,B 0,C 180,E1 -29377.746,E2 -29377.746} C_VEL
LIN {X 0,Y 52.981,Z 526.935,A -85,B 0,C 180,E1 -29388.448,E2 -29388.448} C_VEL
LIN {X 0,Y 46.009,Z 529.373,A -85,B 0,C 180,E1 -29402.722,E2 -29402.722} C_VEL
LIN {X 0,Y 42.281,Z 530.584,A -85,B 0,C 180,E1 -29420.428,E2 -29420.428} C_VEL
LIN {X 0,Y 42.245,Z 530.599,A -85,B 0,C 180,E1 -29439.573,E2 -29439.573} C_VEL
LIN {X 0,Y 45.939,Z 529.423,A -85,B 0,C 180,E1 -29457.316,E2 -29457.316} C_VEL
LIN {X 0,Y 52.933,Z 527.018,A -85,B 0,C 180,E1 -29471.59,E2 -29471.59} C_VEL
LIN {X 0,Y 62.173,Z 523.319,A -85,B 0,C 180,E1 -29482.3,E2 -29482.3} C_VEL
LIN {X 0,Y 73.12,Z 518.208,A -85,B 0,C 180,E1 -29489.882,E2 -29489.882} C_VEL
LIN {X 0,Y 84.767,Z 511.574,A -85,B 0,C 180,E1 -29495.778,E2 -29495.778} C_VEL
LIN {X 0,Y 95.567,Z 504.273,A -85,B 0,C 180,E1 -29499.652,E2 -29499.652} C_VEL
LIN {X 0,Y 106.756,Z 495.36,A -85,B 0,C 180,E1 -29502.655,E2 -29502.655} C_VEL
LIN {X 0,Y 116.484,Z 486.146,A -85,B 0,C 180,E1 -29504.866,E2 -29504.866} C_VEL
LIN {X 0,Y 126.384,Z 475.094,A -85,B 0,C 180,E1 -29506.683,E2 -29506.683} C_VEL
LIN {X 0,Y 134.587,Z 464.128,A -85,B 0,C 180,E1 -29508.068,E2 -29508.068} C_VEL
LIN {X 0,Y 141.348,Z 453.393,A -85,B 0,C 180,E1 -29509.101,E2 -29509.101} C_VEL
LIN {X 0,Y 148.091,Z 440.57,A -85,B 0,C 180,E1 -29509.967,E2 -29509.967} C_VEL
LIN {X 0,Y 153.568,Z 427.476,A -85,B 0,C 180,E1 -29510.671,E2 -29510.671} C_VEL
LIN {X 0,Y 158.167,Z 413.036,A -85,B 0,C 180,E1 -29511.243,E2 -29511.243} C_VEL
LIN {X 0,Y 161.398,Z 398.45,A -85,B 0,C 180,E1 -29511.646,E2 -29511.646} C_VEL
LIN {X 0,Y 164.229,Z 376.752,A -85,B 0,C 180,E1 -29512.056,E2 -29512.056} C_VEL
LIN {X 0,Y 163.755,Z 374.238,A -85,B 0,C 180,E1 -29515.075,E2 -29515.075} C_VEL
LIN {X 0,Y 163.602,Z 373.046,A -85,B 0,C 180,E1 -29517.537,E2 -29517.537} C_VEL
LIN {X 0,Y 163.623,Z 373.285,A -85,B 0,C 180,E1 -29520.615,E2 -29520.615} C_VEL
LIN {X 0,Y 163.833,Z 374.943,A -85,B 0,C 180,E1 -29523.227,E2 -29523.227} C_VEL
LIN {X 0,Y 164.181,Z 377.013,A -85,B 0,C 180,E1 -29525.389,E2 -29525.389} C_VEL
LIN {X 0,Y 161.278,Z 399.3,A -85,B 0,C 180,E1 -29525.796,E2 -29525.796} C_VEL
LIN {X 0,Y 157.971,Z 414.095,A -85,B 0,C 180,E1 -29526.109,E2 -29526.109} C_VEL
LIN {X 0,Y 153.421,Z 428.343,A -85,B 0,C 180,E1 -29526.565,E2 -29526.565} C_VEL
LIN {X 0,Y 147.847,Z 441.644,A -85,B 0,C 180,E1 -29527.125,E2 -29527.125} C_VEL
LIN {X 0,Y 141.003,Z 454.657,A -85,B 0,C 180,E1 -29527.863,E2 -29527.863} C_VEL
LIN {X 0,Y 133.186,Z 466.874,A -85,B 0,C 180,E1 -29528.866,E2 -29528.866} C_VEL
LIN {X 0,Y 124.921,Z 477.745,A -85,B 0,C 180,E1 -29530.099,E2 -29530.099} C_VEL
LIN {X 0,Y 114.875,Z 488.841,A -85,B 0,C 180,E1 -29531.808,E2 -29531.808} C_VEL
LIN {X 0,Y 104.96,Z 498.141,A -85,B 0,C 180,E1 -29533.864,E2 -29533.864} C_VEL
LIN {X 0,Y 93.474,Z 507.278,A -85,B 0,C 180,E1 -29536.92,E2 -29536.92} C_VEL
LIN {X 0,Y 82.707,Z 514.613,A -85,B 0,C 180,E1 -29540.824,E2 -29540.824} C_VEL
LIN {X 0,Y 70.793,Z 521.43,A -85,B 0,C 180,E1 -29546.693,E2 -29546.693} C_VEL
LIN {X 0,Y 59.936,Z 526.708,A -85,B 0,C 180,E1 -29554.84,E2 -29554.84} C_VEL
LIN {X 0,Y 50.713,Z 530.585,A -85,B 0,C 180,E1 -29566.144,E2 -29566.144} C_VEL
LIN {X 0,Y 44.146,Z 533.152,A -85,B 0,C 180,E1 -29581.476,E2 -29581.476} C_VEL
LIN {X 0,Y 41.393,Z 534.466,A -85,B 0,C 180,E1 -29600.228,E2 -29600.228} C_VEL
LIN {X 0,Y 41.51,Z 534.649,A -85,B 0,C 180,E1 -29610.004,E2 -29610.004} C_VEL
LIN {X 0,Y 42.265,Z 533.941,A -85,B 0,C 180,E1 -29629.428,E2 -29629.428} C_VEL
LIN {X 0,Y 47.051,Z 531.974,A -85,B 0,C 180,E1 -29646.693,E2 -29646.693} C_VEL
LIN {X 0,Y 56.013,Z 528.344,A -85,B 0,C 180,E1 -29661.146,E2 -29661.146} C_VEL
LIN {X 0,Y 65.209,Z 524.143,A -85,B 0,C 180,E1 -29669.569,E2 -29669.569} C_VEL
LIN {X 0,Y 76.67,Z 518.079,A -85,B 0,C 180,E1 -29676.444,E2 -29676.444} C_VEL
LIN {X 0,Y 88.747,Z 510.45,A -85,B 0,C 180,E1 -29681.533,E2 -29681.533} C_VEL
LIN {X 0,Y 100.066,Z 501.996,A -85,B 0,C 180,E1 -29684.955,E2 -29684.955} C_VEL
LIN {X 0,Y 111.535,Z 491.82,A -85,B 0,C 180,E1 -29687.604,E2 -29687.604} C_VEL
LIN {X 0,Y 121.56,Z 481.318,A -85,B 0,C 180,E1 -29689.378,E2 -29689.378} C_VEL
LIN {X 0,Y 130.556,Z 470.105,A -85,B 0,C 180,E1 -29690.799,E2 -29690.799} C_VEL
LIN {X 0,Y 138.441,Z 458.423,A -85,B 0,C 180,E1 -29691.861,E2 -29691.861} C_VEL
LIN {X 0,Y 145.279,Z 446.286,A -85,B 0,C 180,E1 -29692.617,E2 -29692.617} C_VEL
LIN {X 0,Y 151.7,Z 432.024,A -85,B 0,C 180,E1 -29693.298,E2 -29693.298} C_VEL
LIN {X 0,Y 156.642,Z 417.704,A -85,B 0,C 180,E1 -29693.773,E2 -29693.773} C_VEL
LIN {X 0,Y 160.25,Z 403.045,A -85,B 0,C 180,E1 -29694.129,E2 -29694.129} C_VEL
LIN {X 0,Y 162.561,Z 387.91,A -85,B 0,C 180,E1 -29694.444,E2 -29694.444} C_VEL
LIN {X 0,Y 163.879,Z 376.595,A -85,B 0,C 180,E1 -29694.685,E2 -29694.685} C_VEL
LIN {X 0,Y 163.424,Z 373.839,A -85,B 0,C 180,E1 -29697.844,E2 -29697.844} C_VEL
LIN {X 0,Y 163.345,Z 373.327,A -85,B 0,C 180,E1 -29698.802,E2 -29698.802} C_VEL
LIN {X 0,Y 163.215,Z 373.782,A -85,B 0,C 180,E1 -29699.487,E2 -29699.487} C_VEL
LIN {X 0,Y 162.841,Z 376.327,A -85,B 0,C 180,E1 -29700.398,E2 -29700.398} C_VEL
LIN {X 0,Y 162.459,Z 379.278,A -85,B 0,C 180,E1 -29701.42,E2 -29701.42} C_VEL
LIN {X 0,Y 162.406,Z 379.79,A -85,B 0,C 180,E1 -29702.019,E2 -29702.019} C_VEL
LIN {X 0,Y 162.456,Z 380.394,A -85,B 0,C 180,E1 -29703.698,E2 -29703.698} C_VEL
LIN {X 0,Y 162.634,Z 381.646,A -85,B 0,C 180,E1 -29705.687,E2 -29705.687} C_VEL
LIN {X 0,Y 159.901,Z 400.881,A -85,B 0,C 180,E1 -29706.008,E2 -29706.008} C_VEL
LIN {X 0,Y 156.458,Z 415.301,A -85,B 0,C 180,E1 -29706.358,E2 -29706.358} C_VEL
LIN {X 0,Y 151.758,Z 429.31,A -85,B 0,C 180,E1 -29706.887,E2 -29706.887} C_VEL
LIN {X 0,Y 146.2,Z 442.042,A -85,B 0,C 180,E1 -29707.489,E2 -29707.489} C_VEL
LIN {X 0,Y 139.348,Z 454.639,A -85,B 0,C 180,E1 -29708.195,E2 -29708.195} C_VEL
LIN {X 0,Y 131.964,Z 465.913,A -85,B 0,C 180,E1 -29709.194,E2 -29709.194} C_VEL
LIN {X 0,Y 123.293,Z 477.003,A -85,B 0,C 180,E1 -29710.487,E2 -29710.487} C_VEL
LIN {X 0,Y 113.187,Z 487.777,A -85,B 0,C 180,E1 -29712.053,E2 -29712.053} C_VEL
LIN {X 0,Y 103.243,Z 496.77,A -85,B 0,C 180,E1 -29714.06,E2 -29714.06} C_VEL
LIN {X 0,Y 93.379,Z 504.37,A -85,B 0,C 180,E1 -29716.338,E2 -29716.338} C_VEL
LIN {X 0,Y 82.14,Z 511.706,A -85,B 0,C 180,E1 -29719.748,E2 -29719.748} C_VEL
LIN {X 0,Y 69.886,Z 518.39,A -85,B 0,C 180,E1 -29725.164,E2 -29725.164} C_VEL
LIN {X 0,Y 58.139,Z 523.542,A -85,B 0,C 180,E1 -29732.198,E2 -29732.198} C_VEL
LIN {X 0,Y 47.895,Z 527.269,A -85,B 0,C 180,E1 -29742.799,E2 -29742.799} C_VEL
LIN {X 0,Y 39.827,Z 529.707,A -85,B 0,C 180,E1 -29758.032,E2 -29758.032} C_VEL
LIN {X 0,Y 35.305,Z 530.917,A -85,B 0,C 180,E1 -29778.513,E2 -29778.513} C_VEL
LIN {X 0,Y 34.727,Z 531.072,A -85,B 0,C 180,E1 -29789.996,E2 -29789.996} C_VEL
LIN {X 0,Y 36.957,Z 530.495,A -85,B 0,C 180,E1 -29812.349,E2 -29812.349} C_VEL
LIN {X 0,Y 43.442,Z 528.711,A -85,B 0,C 180,E1 -29830.32,E2 -29830.32} C_VEL
LIN {X 0,Y 52.778,Z 525.667,A -85,B 0,C 180,E1 -29843.025,E2 -29843.025} C_VEL
LIN {X 0,Y 63.85,Z 521.279,A -85,B 0,C 180,E1 -29851.704,E2 -29851.704} C_VEL
LIN {X 0,Y 72.824,Z 517.018,A -85,B 0,C 180,E1 -29856.457,E2 -29856.457} C_VEL
LIN {X 0,Y 82.104,Z 511.911,A -85,B 0,C 180,E1 -29860.311,E2 -29860.311} C_VEL
LIN {X 0,Y 93.34,Z 504.612,A -85,B 0,C 180,E1 -29863.733,E2 -29863.733} C_VEL
LIN {X 0,Y 104.858,Z 495.708,A -85,B 0,C 180,E1 -29866.363,E2 -29866.363} C_VEL
LIN {X 0,Y 114.837,Z 486.5,A -85,B 0,C 180,E1 -29868.281,E2 -29868.281} C_VEL
LIN {X 0,Y 124.944,Z 475.464,A -85,B 0,C 180,E1 -29869.843,E2 -29869.843} C_VEL
LIN {X 0,Y 133.53,Z 464.2,A -85,B 0,C 180,E1 -29871.079,E2 -29871.079} C_VEL
LIN {X 0,Y 141.038,Z 452.388,A -85,B 0,C 180,E1 -29872.033,E2 -29872.033} C_VEL
LIN {X 0,Y 147.881,Z 439.266,A -85,B 0,C 180,E1 -29872.768,E2 -29872.768} C_VEL
LIN {X 0,Y 153.443,Z 425.743,A -85,B 0,C 180,E1 -29873.365,E2 -29873.365} C_VEL
LIN {X 0,Y 158.007,Z 410.937,A -85,B 0,C 180,E1 -29873.861,E2 -29873.861} C_VEL
LIN {X 0,Y 161.055,Z 396.425,A -85,B 0,C 180,E1 -29874.173,E2 -29874.173} C_VEL
LIN {X 0,Y 162.936,Z 381.899,A -85,B 0,C 180,E1 -29874.451,E2 -29874.451} C_VEL
LIN {X 0,Y 162.733,Z 380.133,A -85,B 0,C 180,E1 -29877.524,E2 -29877.524} C_VEL
LIN {X 0,Y 162.745,Z 380.441,A -85,B 0,C 180,E1 -29880.618,E2 -29880.618} C_VEL
LIN {X 0,Y 162.869,Z 381.777,A -85,B 0,C 180,E1 -29882.636,E2 -29882.636} C_VEL
LIN {X 0,Y 162.904,Z 382.09,A -85,B 0,C 180,E1 -29883.001,E2 -29883.001} C_VEL
LIN {X 0,Y 160.289,Z 400.691,A -85,B 0,C 180,E1 -29883.316,E2 -29883.316} C_VEL
LIN {X 0,Y 156.59,Z 416.213,A -85,B 0,C 180,E1 -29883.59,E2 -29883.59} C_VEL
LIN {X 0,Y 151.902,Z 430.085,A -85,B 0,C 180,E1 -29883.974,E2 -29883.974} C_VEL
LIN {X 0,Y 146.266,Z 442.959,A -85,B 0,C 180,E1 -29884.445,E2 -29884.445} C_VEL
LIN {X 0,Y 139.34,Z 455.672,A -85,B 0,C 180,E1 -29885.053,E2 -29885.053} C_VEL
LIN {X 0,Y 130.721,Z 468.615,A -85,B 0,C 180,E1 -29885.978,E2 -29885.978} C_VEL
LIN {X 0,Y 122.149,Z 479.349,A -85,B 0,C 180,E1 -29887.063,E2 -29887.063} C_VEL
LIN {X 0,Y 111.927,Z 490.125,A -85,B 0,C 180,E1 -29888.536,E2 -29888.536} C_VEL
LIN {X 0,Y 101.798,Z 499.163,A -85,B 0,C 180,E1 -29890.34,E2 -29890.34} C_VEL
LIN {X 0,Y 90.162,Z 507.955,A -85,B 0,C 180,E1 -29893.015,E2 -29893.015} C_VEL
LIN {X 0,Y 80.436,Z 514.273,A -85,B 0,C 180,E1 -29896.041,E2 -29896.041} C_VEL
LIN {X 0,Y 67.871,Z 521.092,A -85,B 0,C 180,E1 -29901.268,E2 -29901.268} C_VEL
LIN {X 0,Y 56.134,Z 526.37,A -85,B 0,C 180,E1 -29908.795,E2 -29908.795} C_VEL
LIN {X 0,Y 45.806,Z 530.248,A -85,B 0,C 180,E1 -29919.908,E2 -29919.908} C_VEL
LIN {X 0,Y 37.992,Z 532.816,A -85,B 0,C 180,E1 -29936.297,E2 -29936.297} C_VEL
LIN {X 0,Y 34.367,Z 534.13,A -85,B 0,C 180,E1 -29958.204,E2 -29958.204} C_VEL
LIN {X 0,Y 34.394,Z 534.315,A -85,B 0,C 180,E1 -29970.004,E2 -29970.004} C_VEL
LIN {X 0,Y 35.605,Z 533.606,A -85,B 0,C 180,E1 -29993.257,E2 -29993.257} C_VEL
LIN {X 0,Y 41.516,Z 531.637,A -85,B 0,C 180,E1 -30012.625,E2 -30012.625} C_VEL
LIN {X 0,Y 51.11,Z 528.259,A -85,B 0,C 180,E1 -30026.633,E2 -30026.633} C_VEL
LIN {X 0,Y 61.877,Z 523.803,A -85,B 0,C 180,E1 -30035.323,E2 -30035.323} C_VEL
LIN {X 0,Y 74.091,Z 517.737,A -85,B 0,C 180,E1 -30041.546,E2 -30041.546} C_VEL
LIN {X 0,Y 85.913,Z 510.634,A -85,B 0,C 180,E1 -30045.795,E2 -30045.795} C_VEL
LIN {X 0,Y 98.448,Z 501.642,A -85,B 0,C 180,E1 -30048.992,E2 -30048.992} C_VEL
LIN {X 0,Y 108.53,Z 493.052,A -85,B 0,C 180,E1 -30050.947,E2 -30050.947} C_VEL
LIN {X 0,Y 118.743,Z 482.85,A -85,B 0,C 180,E1 -30052.473,E2 -30052.473} C_VEL
LIN {X 0,Y 128.831,Z 470.769,A -85,B 0,C 180,E1 -30053.829,E2 -30053.829} C_VEL
LIN {X 0,Y 137.614,Z 457.997,A -85,B 0,C 180,E1 -30054.795,E2 -30054.795} C_VEL
LIN {X 0,Y 144.536,Z 445.823,A -85,B 0,C 180,E1 -30055.421,E2 -30055.421} C_VEL
LIN {X 0,Y 151.035,Z 431.488,A -85,B 0,C 180,E1 -30055.979,E2 -30055.979} C_VEL
LIN {X 0,Y 156.012,Z 417.113,A -85,B 0,C 180,E1 -30056.371,E2 -30056.371} C_VEL
LIN {X 0,Y 159.554,Z 402.803,A -85,B 0,C 180,E1 -30056.666,E2 -30056.666} C_VEL
LIN {X 0,Y 161.875,Z 387.847,A -85,B 0,C 180,E1 -30056.942,E2 -30056.942} C_VEL
LIN {X 0,Y 162.598,Z 381.707,A -85,B 0,C 180,E1 -30057.098,E2 -30057.098} C_VEL
LIN {X 0,Y 162.428,Z 379.871,A -85,B 0,C 180,E1 -30060,E2 -30060} C_VEL
LIN {X 0,Y 162.406,Z 379.79,A -85,B 0,C 180,E1 -30062.019,E2 -30062.019} C_VEL
LIN {X 0,Y 162.34,Z 380.658,A -85,B 0,C 180,E1 -30062.724,E2 -30062.724} C_VEL
LIN {X 0,Y 162.097,Z 383.104,A -85,B 0,C 180,E1 -30063.307,E2 -30063.307} C_VEL
LIN {X 0,Y 161.743,Z 386.215,A -85,B 0,C 180,E1 -30063.599,E2 -30063.599} C_VEL
LIN {X 0,Y 159.557,Z 400.509,A -85,B 0,C 180,E1 -30063.456,E2 -30063.456} C_VEL
LIN {X 0,Y 155.934,Z 415.608,A -85,B 0,C 180,E1 -30063.77,E2 -30063.77} C_VEL
LIN {X 0,Y 151.073,Z 429.845,A -85,B 0,C 180,E1 -30064.223,E2 -30064.223} C_VEL
LIN {X 0,Y 145.448,Z 442.508,A -85,B 0,C 180,E1 -30064.726,E2 -30064.726} C_VEL
LIN {X 0,Y 138.518,Z 455.061,A -85,B 0,C 180,E1 -30065.301,E2 -30065.301} C_VEL
LIN {X 0,Y 130.628,Z 466.836,A -85,B 0,C 180,E1 -30066.178,E2 -30066.178} C_VEL
LIN {X 0,Y 122.203,Z 477.376,A -85,B 0,C 180,E1 -30067.221,E2 -30067.221} C_VEL
LIN {X 0,Y 111.924,Z 488.135,A -85,B 0,C 180,E1 -30068.508,E2 -30068.508} C_VEL
LIN {X 0,Y 101.754,Z 497.119,A -85,B 0,C 180,E1 -30070.185,E2 -30070.185} C_VEL
LIN {X 0,Y 89.961,Z 505.821,A -85,B 0,C 180,E1 -30072.432,E2 -30072.432} C_VEL
LIN {X 0,Y 80.017,Z 512.047,A -85,B 0,C 180,E1 -30074.948,E2 -30074.948} C_VEL
LIN {X 0,Y 67.17,Z 518.727,A -85,B 0,C 180,E1 -30079.663,E2 -30079.663} C_VEL
LIN {X 0,Y 54.686,Z 523.877,A -85,B 0,C 180,E1 -30085.889,E2 -30085.889} C_VEL
LIN {X 0,Y 43.373,Z 527.604,A -85,B 0,C 180,E1 -30095.881,E2 -30095.881} C_VEL
LIN {X 0,Y 34.016,Z 530.039,A -85,B 0,C 180,E1 -30111.692,E2 -30111.692} C_VEL
LIN {X 0,Y 28.407,Z 531.249,A -85,B 0,C 180,E1 -30135.671,E2 -30135.671} C_VEL
LIN {X 0,Y 27.647,Z 531.404,A -85,B 0,C 180,E1 -30149.995,E2 -30149.995} C_VEL
LIN {X 0,Y 30.507,Z 530.828,A -85,B 0,C 180,E1 -30177.429,E2 -30177.429} C_VEL
LIN {X 0,Y 38.305,Z 529.043,A -85,B 0,C 180,E1 -30197.208,E2 -30197.208} C_VEL
LIN {X 0,Y 48.825,Z 526.001,A -85,B 0,C 180,E1 -30209.723,E2 -30209.723} C_VEL
LIN {X 0,Y 60.807,Z 521.612,A -85,B 0,C 180,E1 -30217.605,E2 -30217.605} C_VEL
LIN {X 0,Y 70.278,Z 517.355,A -85,B 0,C 180,E1 -30221.8,E2 -30221.8} C_VEL
LIN {X 0,Y 79.992,Z 512.248,A -85,B 0,C 180,E1 -30225.106,E2 -30225.106} C_VEL
LIN {X 0,Y 91.609,Z 504.95,A -85,B 0,C 180,E1 -30227.988,E2 -30227.988} C_VEL
LIN {X 0,Y 103.417,Z 496.055,A -85,B 0,C 180,E1 -30230.181,E2 -30230.181} C_VEL
LIN {X 0,Y 113.61,Z 486.854,A -85,B 0,C 180,E1 -30231.783,E2 -30231.783} C_VEL
LIN {X 0,Y 123.892,Z 475.833,A -85,B 0,C 180,E1 -30233.067,E2 -30233.067} C_VEL
LIN {X 0,Y 132.5,Z 464.742,A -85,B 0,C 180,E1 -30234.096,E2 -30234.096} C_VEL
LIN {X 0,Y 140.232,Z 452.802,A -85,B 0,C 180,E1 -30234.902,E2 -30234.902} C_VEL
LIN {X 0,Y 147.158,Z 439.722,A -85,B 0,C 180,E1 -30235.503,E2 -30235.503} C_VEL
LIN {X 0,Y 152.787,Z 426.265,A -85,B 0,C 180,E1 -30236.002,E2 -30236.002} C_VEL
LIN {X 0,Y 157.446,Z 411.47,A -85,B 0,C 180,E1 -30236.419,E2 -30236.419} C_VEL
LIN {X 0,Y 160.51,Z 397.272,A -85,B 0,C 180,E1 -30236.687,E2 -30236.687} C_VEL
LIN {X 0,Y 161.87,Z 387.596,A -85,B 0,C 180,E1 -30236.83,E2 -30236.83} C_VEL
LIN {X 0,Y 161.862,Z 387.232,A -85,B 0,C 180,E1 -30237.511,E2 -30237.511} C_VEL
LIN {X 0,Y 161.863,Z 387.503,A -85,B 0,C 180,E1 -30240.462,E2 -30240.462} C_VEL
LIN {X 0,Y 161.865,Z 387.56,A -85,B 0,C 180,E1 -30240.56,E2 -30240.56} C_VEL
LIN {X 0,Y 159.335,Z 403.482,A -85,B 0,C 180,E1 -30240.824,E2 -30240.824} C_VEL
LIN {X 0,Y 155.472,Z 418.472,A -85,B 0,C 180,E1 -30241.024,E2 -30241.024} C_VEL
LIN {X 0,Y 150.261,Z 432.912,A -85,B 0,C 180,E1 -30241.355,E2 -30241.355} C_VEL
LIN {X 0,Y 144.139,Z 446.031,A -85,B 0,C 180,E1 -30241.785,E2 -30241.785} C_VEL
LIN {X 0,Y 136.276,Z 459.473,A -85,B 0,C 180,E1 -30242.331,E2 -30242.331} C_VEL
LIN {X 0,Y 128.433,Z 470.584,A -85,B 0,C 180,E1 -30243.032,E2 -30243.032} C_VEL
LIN {X 0,Y 118.017,Z 482.823,A -85,B 0,C 180,E1 -30244.104,E2 -30244.104} C_VEL
LIN {X 0,Y 107.637,Z 492.981,A -85,B 0,C 180,E1 -30245.325,E2 -30245.325} C_VEL
LIN {X 0,Y 95.624,Z 502.8,A -85,B 0,C 180,E1 -30247.179,E2 -30247.179} C_VEL
LIN {X 0,Y 83.818,Z 510.866,A -85,B 0,C 180,E1 -30249.653,E2 -30249.653} C_VEL
LIN {X 0,Y 72.136,Z 517.55,A -85,B 0,C 180,E1 -30253.037,E2 -30253.037} C_VEL
LIN {X 0,Y 59.236,Z 523.577,A -85,B 0,C 180,E1 -30258.361,E2 -30258.361} C_VEL
LIN {X 0,Y 46.854,Z 528.226,A -85,B 0,C 180,E1 -30266.742,E2 -30266.742} C_VEL
LIN {X 0,Y 36.545,Z 531.356,A -85,B 0,C 180,E1 -30279.721,E2 -30279.721} C_VEL
LIN {X 0,Y 29.121,Z 533.292,A -85,B 0,C 180,E1 -30301.146,E2 -30301.146} C_VEL
LIN {X 0,Y 27.267,Z 533.981,A -85,B 0,C 180,E1 -30330.005,E2 -30330.005} C_VEL
LIN {X 0,Y 29.146,Z 533.269,A -85,B 0,C 180,E1 -30358.839,E2 -30358.839} C_VEL
LIN {X 0,Y 36.561,Z 531.3,A -85,B 0,C 180,E1 -30380.261,E2 -30380.261} C_VEL
LIN {X 0,Y 47.112,Z 528.056,A -85,B 0,C 180,E1 -30393.522,E2 -30393.522} C_VEL
LIN {X 0,Y 59.24,Z 523.465,A -85,B 0,C 180,E1 -30401.645,E2 -30401.645} C_VEL
LIN {X 0,Y 72.141,Z 517.396,A -85,B 0,C 180,E1 -30406.965,E2 -30406.965} C_VEL
LIN {X 0,Y 83.545,Z 510.833,A -85,B 0,C 180,E1 -30410.315,E2 -30410.315} C_VEL
LIN {X 0,Y 95.626,Z 502.564,A -85,B 0,C 180,E1 -30412.834,E2 -30412.834} C_VEL
LIN {X 0,Y 105.912,Z 494.195,A -85,B 0,C 180,E1 -30414.483,E2 -30414.483} C_VEL
LIN {X 0,Y 116.288,Z 484.278,A -85,B 0,C 180,E1 -30415.717,E2 -30415.717} C_VEL
LIN {X 0,Y 126.201,Z 472.954,A -85,B 0,C 180,E1 -30416.808,E2 -30416.808} C_VEL
LIN {X 0,Y 134.533,Z 461.574,A -85,B 0,C 180,E1 -30417.566,E2 -30417.566} C_VEL
LIN {X 0,Y 142.392,Z 448.593,A -85,B 0,C 180,E1 -30418.145,E2 -30418.145} C_VEL
LIN {X 0,Y 148.513,Z 436.126,A -85,B 0,C 180,E1 -30418.569,E2 -30418.569} C_VEL
LIN {X 0,Y 153.767,Z 422.611,A -85,B 0,C 180,E1 -30418.881,E2 -30418.881} C_VEL
LIN {X 0,Y 157.932,Z 408.161,A -85,B 0,C 180,E1 -30419.107,E2 -30419.107} C_VEL
LIN {X 0,Y 160.781,Z 393.166,A -85,B 0,C 180,E1 -30419.334,E2 -30419.334} C_VEL
LIN {X 0,Y 161.56,Z 387.264,A -85,B 0,C 180,E1 -30419.485,E2 -30419.485} C_VEL
LIN {X 0,Y 161.555,Z 386.894,A -85,B 0,C 180,E1 -30422.494,E2 -30422.494} C_VEL
LIN {X 0,Y 161.561,Z 387.307,A -85,B 0,C 180,E1 -30423.223,E2 -30423.223} C_VEL
LIN {X 0,Y 159.557,Z 400.509,A -85,B 0,C 180,E1 -30423.456,E2 -30423.456} C_VEL
LIN {X 0,Y 158.272,Z 406.604,A -85,B 0,C 180,E1 -30423.469,E2 -30423.469} C_VEL
LIN {X 0,Y 155.016,Z 418.588,A -85,B 0,C 180,E1 -30423.032,E2 -30423.032} C_VEL
LIN {X 0,Y 150.881,Z 430.233,A -85,B 0,C 180,E1 -30422.37,E2 -30422.37} C_VEL
LIN {X 0,Y 148.468,Z 435.939,A -85,B 0,C 180,E1 -30422.106,E2 -30422.106} C_VEL
LIN {X 0,Y 144.406,Z 444.315,A -85,B 0,C 180,E1 -30421.987,E2 -30421.987} C_VEL
LIN {X 0,Y 142.933,Z 447.042,A -85,B 0,C 180,E1 -30422.061,E2 -30422.061} C_VEL
LIN {X 0,Y 135.427,Z 459.604,A -85,B 0,C 180,E1 -30422.577,E2 -30422.577} C_VEL
LIN {X 0,Y 126.73,Z 471.559,A -85,B 0,C 180,E1 -30423.413,E2 -30423.413} C_VEL
LIN {X 0,Y 118.041,Z 481.598,A -85,B 0,C 180,E1 -30424.224,E2 -30424.224} C_VEL
LIN {X 0,Y 107.641,Z 491.701,A -85,B 0,C 180,E1 -30425.313,E2 -30425.313} C_VEL
LIN {X 0,Y 95.583,Z 501.416,A -85,B 0,C 180,E1 -30426.959,E2 -30426.959} C_VEL
LIN {X 0,Y 83.585,Z 509.406,A -85,B 0,C 180,E1 -30428.89,E2 -30428.89} C_VEL
LIN {X 0,Y 71.752,Z 515.936,A -85,B 0,C 180,E1 -30431.621,E2 -30431.621} C_VEL
LIN {X 0,Y 61.804,Z 520.471,A -85,B 0,C 180,E1 -30434.85,E2 -30434.85} C_VEL
LIN {X 0,Y 48.798,Z 525.257,A -85,B 0,C 180,E1 -30440.581,E2 -30440.581} C_VEL
LIN {X 0,Y 39.622,Z 527.938,A -85,B 0,C 180,E1 -30447.509,E2 -30447.509} C_VEL
LIN {X 0,Y 28.793,Z 530.372,A -85,B 0,C 180,E1 -30462.918,E2 -30462.918} C_VEL
LIN {X 0,Y 21.613,Z 531.582,A -85,B 0,C 180,E1 -30491.017,E2 -30491.017} C_VEL
LIN {X 0,Y 20.554,Z 531.737,A -85,B 0,C 180,E1 -30509.993,E2 -30509.993} C_VEL
LIN {X 0,Y 24.429,Z 531.16,A -85,B 0,C 180,E1 -30545.119,E2 -30545.119} C_VEL
LIN {X 0,Y 33.888,Z 529.376,A -85,B 0,C 180,E1 -30566.045,E2 -30566.045} C_VEL
LIN {X 0,Y 45.649,Z 526.335,A -85,B 0,C 180,E1 -30577.47,E2 -30577.47} C_VEL
LIN {X 0,Y 58.473,Z 521.945,A -85,B 0,C 180,E1 -30584.046,E2 -30584.046} C_VEL
LIN {X 0,Y 68.387,Z 517.693,A -85,B 0,C 180,E1 -30587.487,E2 -30587.487} C_VEL
LIN {X 0,Y 78.465,Z 512.585,A -85,B 0,C 180,E1 -30590.134,E2 -30590.134} C_VEL
LIN {X 0,Y 90.4,Z 505.289,A -85,B 0,C 180,E1 -30592.389,E2 -30592.389} C_VEL
LIN {X 0,Y 102.447,Z 496.401,A -85,B 0,C 180,E1 -30594.087,E2 -30594.087} C_VEL
LIN {X 0,Y 112.816,Z 487.207,A -85,B 0,C 180,E1 -30595.345,E2 -30595.345} C_VEL
LIN {X 0,Y 123.238,Z 476.201,A -85,B 0,C 180,E1 -30596.334,E2 -30596.334} C_VEL
LIN {X 0,Y 132.802,Z 463.963,A -85,B 0,C 180,E1 -30597.247,E2 -30597.247} C_VEL
LIN {X 0,Y 140.655,Z 451.764,A -85,B 0,C 180,E1 -30597.844,E2 -30597.844} C_VEL
LIN {X 0,Y 147.647,Z 438.338,A -85,B 0,C 180,E1 -30598.322,E2 -30598.322} C_VEL
LIN {X 0,Y 147.618,Z 438.416,A -85,B 0,C 180,E1 -30598.765,E2 -30598.765} C_VEL
LIN {X 0,Y 140.572,Z 451.952,A -85,B 0,C 180,E1 -30599.11,E2 -30599.11} C_VEL
LIN {X 0,Y 131.774,Z 465.468,A -85,B 0,C 180,E1 -30599.581,E2 -30599.581} C_VEL
LIN {X 0,Y 122.218,Z 477.497,A -85,B 0,C 180,E1 -30600.293,E2 -30600.293} C_VEL
LIN {X 0,Y 112.463,Z 487.769,A -85,B 0,C 180,E1 -30601.055,E2 -30601.055} C_VEL
LIN {X 0,Y 101.968,Z 497.095,A -85,B 0,C 180,E1 -30602.07,E2 -30602.07} C_VEL
LIN {X 0,Y 89.78,Z 506.133,A -85,B 0,C 180,E1 -30603.597,E2 -30603.597} C_VEL
LIN {X 0,Y 77.701,Z 513.592,A -85,B 0,C 180,E1 -30605.791,E2 -30605.791} C_VEL
LIN {X 0,Y 64.073,Z 520.416,A -85,B 0,C 180,E1 -30609.199,E2 -30609.199} C_VEL
LIN {X 0,Y 50.796,Z 525.697,A -85,B 0,C 180,E1 -30614.436,E2 -30614.436} C_VEL
LIN {X 0,Y 38.219,Z 529.577,A -85,B 0,C 180,E1 -30623.169,E2 -30623.169} C_VEL
LIN {X 0,Y 27.237,Z 532.143,A -85,B 0,C 180,E1 -30639.287,E2 -30639.287} C_VEL
LIN {X 0,Y 20.571,Z 533.459,A -85,B 0,C 180,E1 -30670.031,E2 -30670.031} C_VEL
LIN {X 0,Y 20.159,Z 533.647,A -85,B 0,C 180,E1 -30690.007,E2 -30690.007} C_VEL
LIN {X 0,Y 23.124,Z 532.932,A -85,B 0,C 180,E1 -30727.442,E2 -30727.442} C_VEL
LIN {X 0,Y 32.45,Z 530.964,A -85,B 0,C 180,E1 -30750.04,E2 -30750.04} C_VEL
LIN {X 0,Y 44.376,Z 527.718,A -85,B 0,C 180,E1 -30761.857,E2 -30761.857} C_VEL
LIN {X 0,Y 57.379,Z 523.124,A -85,B 0,C 180,E1 -30768.493,E2 -30768.493} C_VEL
LIN {X 0,Y 70.867,Z 517.055,A -85,B 0,C 180,E1 -30772.631,E2 -30772.631} C_VEL
LIN {X 0,Y 81.826,Z 510.971,A -85,B 0,C 180,E1 -30775.074,E2 -30775.074} C_VEL
LIN {X 0,Y 93.259,Z 503.458,A -85,B 0,C 180,E1 -30776.902,E2 -30776.902} C_VEL
LIN {X 0,Y 105.464,Z 493.837,A -85,B 0,C 180,E1 -30778.358,E2 -30778.358} C_VEL
LIN {X 0,Y 115.973,Z 483.909,A -85,B 0,C 180,E1 -30779.238,E2 -30779.238} C_VEL
LIN {X 0,Y 125.174,Z 473.585,A -85,B 0,C 180,E1 -30780.001,E2 -30780.001} C_VEL
LIN {X 0,Y 134.419,Z 461.163,A -85,B 0,C 180,E1 -30780.611,E2 -30780.611} C_VEL
LIN {X 0,Y 142.34,Z 448.148,A -85,B 0,C 180,E1 -30781.011,E2 -30781.011} C_VEL
LIN {X 0,Y 147.625,Z 437.621,A -85,B 0,C 180,E1 -30781.271,E2 -30781.271} C_VEL
LIN {X 0,Y 147.659,Z 437.531,A -85,B 0,C 180,E1 -30781.767,E2 -30781.767} C_VEL
LIN {X 0,Y 142.933,Z 447.042,A -85,B 0,C 180,E1 -30782.061,E2 -30782.061} C_VEL
LIN {X 0,Y 142.679,Z 448.024,A -85,B 0,C 180,E1 -30782.079,E2 -30782.079} C_VEL
LIN {X 0,Y 142.679,Z 509.328,A -85,B 0,C 180,E1 -30782.079,E2 -30782.079} C_VEL
LIN {X 0,Y 103.644,Z 509.328,A -85,B 0,C 180,E1 -30782.057,E2 -30782.057} C_VEL
LIN {X 0,Y 101.644,Z 507.328,A -85,B 0,C 180,E1 -30782.055,E2 -30782.055} C_VEL
LIN {X 0,Y 101.644,Z 500.754,A -85,B 0,C 180,E1 -30782.055,E2 -30782.055} C_VEL
LIN {X 0,Y 98.476,Z 499.161,A -85,B 0,C 180,E1 -30782.344,E2 -30782.344} C_VEL
LIN {X 0,Y 86.262,Z 507.613,A -85,B 0,C 180,E1 -30783.574,E2 -30783.574} C_VEL
LIN {X 0,Y 72.854,Z 515.173,A -85,B 0,C 180,E1 -30785.537,E2 -30785.537} C_VEL
LIN {X 0,Y 60.377,Z 520.807,A -85,B 0,C 180,E1 -30788.33,E2 -30788.33} C_VEL
LIN {X 0,Y 46.777,Z 525.591,A -85,B 0,C 180,E1 -30792.412,E2 -30792.412} C_VEL
LIN {X 0,Y 36.88,Z 528.272,A -85,B 0,C 180,E1 -30797.658,E2 -30797.658} C_VEL
LIN {X 0,Y 24.513,Z 530.705,A -85,B 0,C 180,E1 -30810.662,E2 -30810.662} C_VEL
LIN {X 0,Y 15.079,Z 531.915,A -85,B 0,C 180,E1 -30842.209,E2 -30842.209} C_VEL
LIN {X 0,Y 13.481,Z 532.069,A -85,B 0,C 180,E1 -30869.989,E2 -30869.989} C_VEL
LIN {X 0,Y 19.075,Z 531.492,A -85,B 0,C 180,E1 -30917.455,E2 -30917.455} C_VEL
LIN {X 0,Y 30.495,Z 529.708,A -85,B 0,C 180,E1 -30937.186,E2 -30937.186} C_VEL
LIN {X 0,Y 43.421,Z 526.669,A -85,B 0,C 180,E1 -30946.184,E2 -30946.184} C_VEL
LIN {X 0,Y 56.933,Z 522.278,A -85,B 0,C 180,E1 -30950.926,E2 -30950.926} C_VEL
LIN {X 0,Y 70.646,Z 516.442,A -85,B 0,C 180,E1 -30954.137,E2 -30954.137} C_VEL
LIN {X 0,Y 82.014,Z 510.392,A -85,B 0,C 180,E1 -30955.953,E2 -30955.953} C_VEL
LIN {X 0,Y 94.971,Z 502.014,A -85,B 0,C 180,E1 -30957.408,E2 -30957.408} C_VEL
LIN {X 0,Y 98.465,Z 499.434,A -85,B 0,C 180,E1 -30957.739,E2 -30957.739} C_VEL
LIN {X 0,Y 98.432,Z 499.48,A -85,B 0,C 180,E1 -30958.293,E2 -30958.293} C_VEL
LIN {X 0,Y 86.094,Z 508.051,A -85,B 0,C 180,E1 -30959.379,E2 -30959.379} C_VEL
LIN {X 0,Y 73.801,Z 515.089,A -85,B 0,C 180,E1 -30960.974,E2 -30960.974} C_VEL
LIN {X 0,Y 59.847,Z 521.529,A -85,B 0,C 180,E1 -30963.506,E2 -30963.506} C_VEL
LIN {X 0,Y 46.079,Z 526.453,A -85,B 0,C 180,E1 -30967.56,E2 -30967.56} C_VEL
LIN {X 0,Y 36.002,Z 529.24,A -85,B 0,C 180,E1 -30972.585,E2 -30972.585} C_VEL
LIN {X 0,Y 23.365,Z 531.807,A -85,B 0,C 180,E1 -30985.545,E2 -30985.545} C_VEL
LIN {X 0,Y 14.052,Z 533.123,A -85,B 0,C 180,E1 -31020.002,E2 -31020.002} C_VEL
LIN {X 0,Y 13.018,Z 533.312,A -85,B 0,C 180,E1 -31050.011,E2 -31050.011} C_VEL
LIN {X 0,Y 17.974,Z 532.596,A -85,B 0,C 180,E1 -31101.459,E2 -31101.459} C_VEL
LIN {X 0,Y 29.523,Z 530.626,A -85,B 0,C 180,E1 -31122.231,E2 -31122.231} C_VEL
LIN {X 0,Y 42.688,Z 527.38,A -85,B 0,C 180,E1 -31131.065,E2 -31131.065} C_VEL
LIN {X 0,Y 56.387,Z 522.785,A -85,B 0,C 180,E1 -31135.671,E2 -31135.671} C_VEL
LIN {X 0,Y 70.307,Z 516.713,A -85,B 0,C 180,E1 -31138.457,E2 -31138.457} C_VEL
LIN {X 0,Y 82.636,Z 509.979,A -85,B 0,C 180,E1 -31140.234,E2 -31140.234} C_VEL
LIN {X 0,Y 94.91,Z 501.863,A -85,B 0,C 180,E1 -31141.464,E2 -31141.464} C_VEL
LIN {X 0,Y 98.437,Z 499.214,A -85,B 0,C 180,E1 -31141.716,E2 -31141.716} C_VEL
LIN {X 0,Y 98.476,Z 499.161,A -85,B 0,C 180,E1 -31142.344,E2 -31142.344} C_VEL
LIN {X 0,Y 98.584,Z 501.158,A -85,B 0,C 180,E1 -31143.563,E2 -31143.563} C_VEL
LIN {X 0,Y 98.584,Z 534.576,A -85,B 0,C 180,E1 -31143.563,E2 -31143.563} C_VEL
LIN {X 0,Y 53.805,Z 534.576,A -85,B 0,C 180,E1 -31142.67,E2 -31142.67} C_VEL
LIN {X 0,Y 51.806,Z 532.576,A -85,B 0,C 180,E1 -31142.594,E2 -31142.594} C_VEL
LIN {X 0,Y 51.806,Z 526.796,A -85,B 0,C 180,E1 -31142.594,E2 -31142.594} C_VEL
LIN {X 0,Y 49.267,Z 524.879,A -85,B 0,C 180,E1 -31143.029,E2 -31143.029} C_VEL
LIN {X 0,Y 35.378,Z 528.606,A -85,B 0,C 180,E1 -31146.622,E2 -31146.622} C_VEL
LIN {X 0,Y 21.768,Z 531.038,A -85,B 0,C 180,E1 -31154.382,E2 -31154.382} C_VEL
LIN {X 0,Y 9.413,Z 532.247,A -85,B 0,C 180,E1 -31181.68,E2 -31181.68} C_VEL
LIN {X 0,Y 6.397,Z 532.401,A -85,B 0,C 180,E1 -31229.977,E2 -31229.977} C_VEL
LIN {X 0,Y 15.203,Z 531.825,A -85,B 0,C 180,E1 -31297.571,E2 -31297.571} C_VEL
LIN {X 0,Y 28.501,Z 530.042,A -85,B 0,C 180,E1 -31310.486,E2 -31310.486} C_VEL
LIN {X 0,Y 42.29,Z 527.003,A -85,B 0,C 180,E1 -31315.591,E2 -31315.591} C_VEL
LIN {X 0,Y 49.259,Z 524.983,A -85,B 0,C 180,E1 -31317.034,E2 -31317.034} C_VEL
LIN {X 0,Y 49.223,Z 525.022,A -85,B 0,C 180,E1 -31318,E2 -31318} C_VEL
LIN {X 0,Y 35.143,Z 528.903,A -85,B 0,C 180,E1 -31321.077,E2 -31321.077} C_VEL
LIN {X 0,Y 21.281,Z 531.471,A -85,B 0,C 180,E1 -31327.857,E2 -31327.857} C_VEL
LIN {X 0,Y 8.633,Z 532.788,A -85,B 0,C 180,E1 -31355.538,E2 -31355.538} C_VEL
LIN {X 0,Y 5.891,Z 532.978,A -85,B 0,C 180,E1 -31410.025,E2 -31410.025} C_VEL
LIN {X 0,Y 14.624,Z 532.26,A -85,B 0,C 180,E1 -31484.018,E2 -31484.018} C_VEL
LIN {X 0,Y 28.173,Z 530.288,A -85,B 0,C 180,E1 -31496.308,E2 -31496.308} C_VEL
LIN {X 0,Y 42.174,Z 527.042,A -85,B 0,C 180,E1 -31500.748,E2 -31500.748} C_VEL
LIN {X 0,Y 49.228,Z 524.921,A -85,B 0,C 180,E1 -31502.003,E2 -31502.003} C_VEL
LIN {X 0,Y 49.267,Z 524.879,A -85,B 0,C 180,E1 -31503.029,E2 -31503.029} C_VEL
LIN {X 0,Y 49.422,Z 526.877,A -85,B 0,C 180,E1 -31505.455,E2 -31505.455} C_VEL
LIN {X 0,Y 49.422,Z 600,A -85,B 0,C 180,E1 -31505.455,E2 -31505.455} C_VEL
LIN {X 0,Y 49.422,Z 600,A -85,B 0,C 180,E1 -31505.455,E2 -31505.455}

QRS_NEXT_CUT()

QRS_NEXT()
QRS_HOME()

END
